ABB RobotStudio station: Train Assembling.rspag

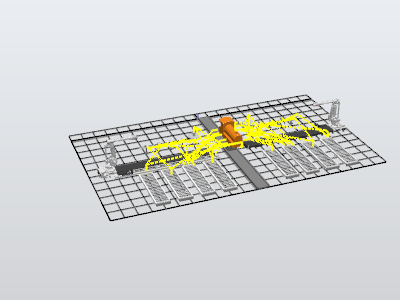
--- station ---
Station SimulationProject (saved by RobotStudio 24.3.10958.1)
Controller SimulationProject, task T_ROB2: task frame (RAPID world) sits at (6025, -9409.5, 384.5) mm, rotated rx 0 ry 0 rz 90 deg in the station
Controller SimulationProject, task T_ROB1: task frame (RAPID world) sits at (6025, -9409.5, 384.5) mm, rotated rx 0 ry 0 rz 90 deg in the station
Controller SimulationProject
  mechanical unit ROB_1: IRB6660_100_335__01_R, 6 joints, base frame (0, 0, 0) mm
  mechanical unit TRACK_1: IRBT6004_STD_0_0_8__04_R, 1 joints, base frame (0, 0, 0) mm
  mechanical unit ROB_2: IRB6660_100_335__01_L, 6 joints, base frame (19319, 50, 0) mm, rotated rx 0 ry 0 rz 180 deg
  mechanical unit TRACK_2: IRBT6004_STD_0_0_8__04_L, 1 joints, base frame (19319, 50, 0) mm, rotated rx 0 ry 0 rz 180 deg
Layout (positions relative to the parent item):
  - IRB6660_100_335__01_R [mechanism, from %ABB.RobotStudio.Models.IRB6660%\IRB6660_100_335_G_01.rslib] at (6025, -9409.5, 384.5) mm, rotated rx 0 ry 0 rz 90 deg; joint values [0, 0, 0, 0, 0.5236, 0] (rad or m)
  - IRBT6004_STD_0_0_8__04_R [mechanism] at (6500, -10000, 0) mm, rotated rx 0 ry 0 rz 90 deg; joint values [0] (rad or m)
      links: Base, Link1
  - IRB6660_100_335__01_L [mechanism, from %ABB.RobotStudio.Models.IRB6660%\IRB6660_100_335_G_01.rslib] at (5975, 9909.5, 384.5) mm, rotated rx 0 ry 0 rz -90 deg; joint values [0, 0, 0, 0, 0.5236, 0] (rad or m)
  - IRBT6004_STD_0_0_8__04_L [mechanism] at (5500, 10500, 0) mm, rotated rx 0 ry 0 rz -90 deg; joint values [0] (rad or m)
      links: Base, Link1
  - Train_Slider_Device [mechanism, from Tools\Train_Slider_Device.rslib] at (0, 0, 0) mm; joint values [5.8] (rad or m)
  - train_body [part] at (4625, 0, 1000) mm, rotated rx 90 ry 0 rz 90 deg, size 1000 x 1362.5 x 2750 mm
  - SC_Wheel_InFeeder_R [smart component]
      signals: DI FeedWheel
      connections:
        SC_Wheel_InFeeder_R.FeedWheel -> Source.Execute
        Source.Executed -> Queue.Enqueue
        PlaneSensor.SensorOut -> Queue.Dequeue
        Source.Copy => Queue.Back
        Queue.Front => PlaneSensor.SensedPart
    - LinearMover [smart component, from Components\LinearMover.rslib]
        properties: Object=Queue; Direction=[-1 0 0]; Speed=0.5; Reference=Global; ReferenceObject=(none)
    - Source [smart component, from Components\Source.rslib]
        properties: Source=Wheel_R; Copy=(none); Parent=(none); Position=[0 0 0]; Orientation=[0 0 0]; Transient=false; PhysicsBehavior=-1
    - Queue [smart component, from Components\Queue.rslib]
        properties: Back=(none); Front=(none); Queue={9305e1b5-9379-48da-9073-8e46354b7aa1};{06ef701b-e628-484b-9ba1-8a04eedeb4da};{5bc8af88-7b1d-4971-8da9-7f0ec308ea46};{a84a56de-22f5-4cb1-84ca-754a15d204a5};{2fea0387-14bd-40cc-a5c2-ab10d6d0a730};{1b48ac47-8c9f-46e7-a90e-52eff258e1c6};{a66a5858-2d20-4f19-907b-7c595a4e8944}; NumberOfObjects=1
    - PlaneSensor [smart component, from Components\PlaneSensor.rslib]
        properties: Origin=[7.64 -1.525 0.435]; Axis1=[0 0 0.2]; Axis2=[0 -0.9 0]; Tag=(none); SensedPart=(none)
      - _sensorPart_ [part], size 0 x 900 x 200 mm
    - InFeeder_R_1 [part] at (6500, -2000, 0) mm, size 4244 x 1170 x 435 mm
  - SC_Screws_InFeeder_R [smart component]
      signals: DI FeedScrews
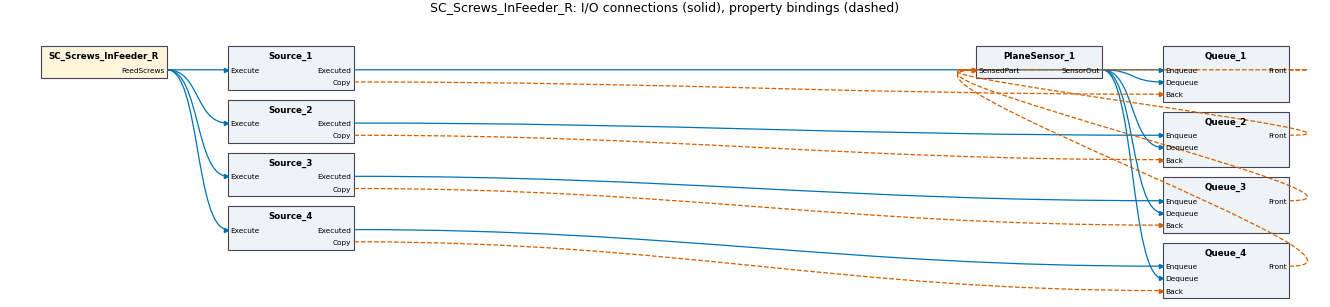
      connections:
        Source_1.Executed -> Queue_1.Enqueue
        Source_2.Executed -> Queue_2.Enqueue
        PlaneSensor_1.SensorOut -> Queue_1.Dequeue
        PlaneSensor_1.SensorOut -> Queue_2.Dequeue
        Source_3.Executed -> Queue_3.Enqueue
        Source_4.Executed -> Queue_4.Enqueue
        PlaneSensor_1.SensorOut -> Queue_3.Dequeue
        PlaneSensor_1.SensorOut -> Queue_4.Dequeue
        SC_Screws_InFeeder_R.FeedScrews -> Source_1.Execute
        SC_Screws_InFeeder_R.FeedScrews -> Source_2.Execute
        SC_Screws_InFeeder_R.FeedScrews -> Source_3.Execute
        SC_Screws_InFeeder_R.FeedScrews -> Source_4.Execute
        Source_1.Copy => Queue_1.Back
        Queue_1.Front => PlaneSensor_1.SensedPart
        Queue_2.Front => PlaneSensor_1.SensedPart
        Source_3.Copy => Queue_3.Back
        Source_4.Copy => Queue_4.Back
        Queue_3.Front => PlaneSensor_1.SensedPart
        Queue_4.Front => PlaneSensor_1.SensedPart
        Source_2.Copy => Queue_2.Back
    - InFeeder_R_2 [part] at (6500, -3700, 0) mm, size 4244 x 1170 x 435 mm
    - Source_1 [smart component, from Components\Source.rslib]
        properties: Source=Axel_pin_R_1; Copy=(none); Parent=(none); Position=[0 0 0]; Orientation=[0 0 0]; Transient=false; PhysicsBehavior=-1
    - Source_2 [smart component, from Components\Source.rslib]
        properties: Source=Axel_pin_R_2; Copy=(none); Parent=(none); Position=[0 0 0]; Orientation=[0 0 0]; Transient=false; PhysicsBehavior=-1
    - PlaneSensor_1 [smart component, from Components\PlaneSensor.rslib]
        properties: Origin=[7.64 -3.225 0.435]; Axis1=[0 -0.9 0]; Axis2=[0 0 0.2]; Tag=(none); SensedPart=(none)
      - _sensorPart_ [part], size 0 x 900 x 200 mm
    - Queue_1 [smart component, from Components\Queue.rslib]
        properties: Back=(none); Front=(none); Queue={97678c5a-5102-4407-a08a-453d650fad80};{250eec11-255d-4adc-99c6-b5c3b0be1ee0};{db8d0e62-9b7f-46e3-aee1-3fad0f8208f2};{3d23516b-ce9b-4da7-b7d3-33ea277e23c2};{336e8d4f-087f-4f39-84d7-9a0945deb51c};{844237c7-2bfb-4aaa-a27e-a2dee6dfaffc};{404c0b62-1524-42dd-8a4b-c3c094d3b07c}; NumberOfObjects=1
    - Queue_2 [smart component, from Components\Queue.rslib]
        properties: Back=(none); Front=(none); Queue={9e77e015-2590-4be3-ac1b-ed1168efcc9a};{9dcada67-6f7e-4e2e-9580-51d109b5ace8};{683b0bf4-25e8-4e74-bd3c-a3e39548362f}; NumberOfObjects=1
    - LinearMover_1 [smart component, from Components\LinearMover.rslib]
        properties: Object=Queue_1; Direction=[-1 0 0]; Speed=0.5; Reference=Global; ReferenceObject=(none)
    - LinearMover_2 [smart component, from Components\LinearMover.rslib]
        properties: Object=Queue_2; Direction=[-1 0 0]; Speed=0.5; Reference=Global; ReferenceObject=(none)
    - Source_3 [smart component, from Components\Source.rslib]
        properties: Source=Arm_pin_R_1; Copy=(none); Parent=(none); Position=[0 0 0]; Orientation=[0 0 0]; Transient=false; PhysicsBehavior=-1
    - Source_4 [smart component, from Components\Source.rslib]
        properties: Source=Arm_pin_R_2; Copy=(none); Parent=(none); Position=[0 0 0]; Orientation=[0 0 0]; Transient=false; PhysicsBehavior=-1
    - Queue_3 [smart component, from Components\Queue.rslib]
        properties: Back=(none); Front=(none); Queue={6ed0c4d3-6d0d-466e-bc0a-e55b9d8fea7f};{e0375d21-1e9d-4950-9f28-cd2b8b21485b};{fc4e43e4-3199-411d-82b8-a28eed2363bc};{00cf09c5-e1bb-4b7d-8b4f-d00f571ac579}; NumberOfObjects=1
    - Queue_4 [smart component, from Components\Queue.rslib]
        properties: Back=(none); Front=(none); Queue={3f8a16d5-ca92-48d5-91d9-dae51837d5b3};{1a52513d-85f7-411d-a240-a53d51e62410};{d2420088-7648-42ee-ace7-0250b97bbbd5};{92784dae-7df1-4f9f-a001-3219d183c38a}; NumberOfObjects=1
    - LinearMover_3 [smart component, from Components\LinearMover.rslib]
        properties: Object=Queue_3; Direction=[-1 0 0]; Speed=0.5; Reference=Global; ReferenceObject=(none)
    - LinearMover_4 [smart component, from Components\LinearMover.rslib]
        properties: Object=Queue_4; Direction=[-1 0 0]; Speed=0.5; Reference=Global; ReferenceObject=(none)
  - SC_Link_InFeeder_R [smart component]
      signals: DI FeedLink
      connections:
        PlaneSensor.SensorOut -> Queue.Dequeue
        Source.Executed -> Queue.Enqueue
        SC_Link_InFeeder_R.FeedLink -> Source.Execute
        Source.Copy => Queue.Back
        Queue.Front => PlaneSensor.SensedPart
    - InFeeder_R_3 [part] at (6500, -5400, 0) mm, size 4244 x 1170 x 435 mm
    - Source [smart component, from Components\Source.rslib]
        properties: Source=Link_R; Copy=(none); Parent=(none); Position=[0 0 0]; Orientation=[0 0 0]; Transient=false; PhysicsBehavior=-1
    - PlaneSensor [smart component, from Components\PlaneSensor.rslib]
        properties: Origin=[7.64 -4.925 0.435]; Axis1=[0 -0.9 0]; Axis2=[0 0 0.2]; Tag=(none); SensedPart=(none)
      - _sensorPart_ [part], size 0 x 900 x 200 mm
    - Queue [smart component, from Components\Queue.rslib]
        properties: Back=(none); Front=(none); Queue={c123ca29-f25a-4360-8441-2d47dce9963e};{cf207c4b-303d-438f-b968-cd8524d1301f};{72cfc707-1568-4af6-a666-0a4982008e72};{3a86617a-4034-4a56-87a3-25b6863a3576}; NumberOfObjects=1
    - LinearMover [smart component, from Components\LinearMover.rslib]
        properties: Object=Queue; Direction=[-1 0 0]; Speed=0.5; Reference=Global; ReferenceObject=(none)
  - SC_CowCatcher_InFeeder_R [smart component]
      signals: DI FeedCowCatcher
      connections:
        SC_CowCatcher_InFeeder_R.FeedCowCatcher -> Source_2.Execute
        Source_2.Executed -> Queue_2.Enqueue
        PlaneSensor_2.SensorOut -> Queue_2.Dequeue
        Source_2.Copy => Queue_2.Back
        Queue_2.Front => PlaneSensor_2.SensedPart
    - InFeeder_R_4 [part] at (6500, -7100, 0) mm, size 4244 x 1170 x 435 mm
    - LinearMover_2 [smart component, from Components\LinearMover.rslib]
        properties: Object=Queue_2; Direction=[-1 0 0]; Speed=0.5; Reference=Global; ReferenceObject=(none)
    - Queue_2 [smart component, from Components\Queue.rslib]
        properties: Back=(none); Front=(none); Queue={e25ade14-9086-4660-97fb-0c3a861d3266};{c5b81c7c-9b40-4532-81d4-bb342586ee21};{586fb502-498d-41ec-904b-685c852027eb}; NumberOfObjects=1
    - PlaneSensor_2 [smart component, from Components\PlaneSensor.rslib]
        properties: Origin=[7.64 -6.625 0.435]; Axis1=[0 -0.9 0]; Axis2=[0 0 0.2]; Tag=(none); SensedPart=(none)
      - _sensorPart_ [part], size 0 x 900 x 200 mm
    - Source_2 [smart component, from Components\Source.rslib]
        properties: Source=Cow_Catcher; Copy=(none); Parent=(none); Position=[0 0 0]; Orientation=[0 0 0]; Transient=false; PhysicsBehavior=-1
  - SC_Link_InFeeder_L [smart component] at (0, 11800, 0) mm
      signals: DI FeedLink_L
      connections:
        PlaneSensor.SensorOut -> Queue.Dequeue
        Source.Executed -> Queue.Enqueue
        SC_Link_InFeeder_L.FeedLink_L -> Source.Execute
        Source.Copy => Queue.Back
        Queue.Front => PlaneSensor.SensedPart
    - InFeeder_R_3 [part] at (6500, -5400, 0) mm, size 4244 x 1170 x 435 mm
    - Source [smart component, from Components\Source.rslib]
        properties: Source=Link_L; Copy=(none); Parent=(none); Position=[0 0 0]; Orientation=[0 0 0]; Transient=false; PhysicsBehavior=-1
    - PlaneSensor [smart component, from Components\PlaneSensor.rslib]
        properties: Origin=[7.64 -4.925 0.435]; Axis1=[0 -0.9 0]; Axis2=[0 0 0.2]; Tag=(none); SensedPart=(none)
      - _sensorPart_ [part], size 0 x 900 x 200 mm
    - Queue [smart component, from Components\Queue.rslib]
        properties: Back=(none); Front=(none); Queue={9254929b-264a-4685-b6a1-bce98a06c028};{c123ca29-f25a-4360-8441-2d47dce9963e};{cf207c4b-303d-438f-b968-cd8524d1301f};{4bafc17b-eeca-41b5-b438-7a43c40b0997};{fc8fee30-79e4-4b7d-9fd5-4bdb28a1c232};{eefd66af-0d0b-49de-8bd5-7017a8631d51};{a98b3633-ee36-4176-97fc-4a52fb264d0f}; NumberOfObjects=1
    - LinearMover [smart component, from Components\LinearMover.rslib]
        properties: Object=Queue; Direction=[-1 0 0]; Speed=0.5; Reference=Global; ReferenceObject=(none)
  - SC_Screws_InFeeder_L [smart component] at (0, 8400, 0) mm
      signals: DI FeedScrews_L
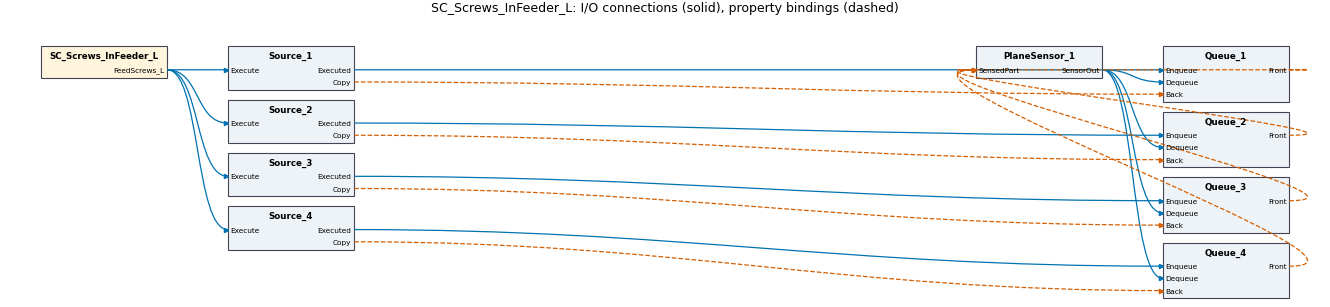
      connections:
        Source_1.Executed -> Queue_1.Enqueue
        Source_2.Executed -> Queue_2.Enqueue
        PlaneSensor_1.SensorOut -> Queue_1.Dequeue
        PlaneSensor_1.SensorOut -> Queue_2.Dequeue
        Source_3.Executed -> Queue_3.Enqueue
        Source_4.Executed -> Queue_4.Enqueue
        PlaneSensor_1.SensorOut -> Queue_3.Dequeue
        PlaneSensor_1.SensorOut -> Queue_4.Dequeue
        SC_Screws_InFeeder_L.FeedScrews_L -> Source_1.Execute
        SC_Screws_InFeeder_L.FeedScrews_L -> Source_2.Execute
        SC_Screws_InFeeder_L.FeedScrews_L -> Source_3.Execute
        SC_Screws_InFeeder_L.FeedScrews_L -> Source_4.Execute
        Source_1.Copy => Queue_1.Back
        Queue_1.Front => PlaneSensor_1.SensedPart
        Queue_2.Front => PlaneSensor_1.SensedPart
        Source_3.Copy => Queue_3.Back
        Source_4.Copy => Queue_4.Back
        Queue_3.Front => PlaneSensor_1.SensedPart
        Queue_4.Front => PlaneSensor_1.SensedPart
        Source_2.Copy => Queue_2.Back
    - InFeeder_R_2 [part] at (6500, -3700, 0) mm, size 4244 x 1170 x 435 mm
    - Source_1 [smart component, from Components\Source.rslib]
        properties: Source=Axel_pin_L_1; Copy=(none); Parent=(none); Position=[0 0 0]; Orientation=[0 0 0]; Transient=false; PhysicsBehavior=-1
    - Source_2 [smart component, from Components\Source.rslib]
        properties: Source=Axel_pin_L_2; Copy=(none); Parent=(none); Position=[0 0 0]; Orientation=[0 0 0]; Transient=false; PhysicsBehavior=-1
    - PlaneSensor_1 [smart component, from Components\PlaneSensor.rslib]
        properties: Origin=[7.64 -3.225 0.435]; Axis1=[0 -0.9 0]; Axis2=[0 0 0.2]; Tag=(none); SensedPart=(none)
      - _sensorPart_ [part], size 0 x 900 x 200 mm
    - Queue_1 [smart component, from Components\Queue.rslib]
        properties: Back=(none); Front=(none); Queue={14a08090-38d6-472e-a98c-ca0218ab0c7a};{97678c5a-5102-4407-a08a-453d650fad80};{250eec11-255d-4adc-99c6-b5c3b0be1ee0};{db8d0e62-9b7f-46e3-aee1-3fad0f8208f2};{2b439d8e-8bb8-4235-883a-6f3a83c8853b};{c95d82af-f454-4449-b05f-7ed691318b29};{bee60a8c-c6b8-489c-bade-25b0cdd1ce0b};{754e9011-9557-4989-aa10-6dc2dc1ac779}; NumberOfObjects=1
    - Queue_2 [smart component, from Components\Queue.rslib]
        properties: Back=(none); Front=(none); Queue=; NumberOfObjects=0
    - LinearMover_1 [smart component, from Components\LinearMover.rslib]
        properties: Object=Queue_1; Direction=[-1 0 0]; Speed=0.5; Reference=Global; ReferenceObject=(none)
    - LinearMover_2 [smart component, from Components\LinearMover.rslib]
        properties: Object=Queue_2; Direction=[-1 0 0]; Speed=0.5; Reference=Global; ReferenceObject=(none)
    - Source_3 [smart component, from Components\Source.rslib]
        properties: Source=Arm_pin_L_1; Copy=(none); Parent=(none); Position=[0 0 0]; Orientation=[0 0 0]; Transient=false; PhysicsBehavior=-1
    - Source_4 [smart component, from Components\Source.rslib]
        properties: Source=Arm_pin_L_2; Copy=(none); Parent=(none); Position=[0 0 0]; Orientation=[0 0 0]; Transient=false; PhysicsBehavior=-1
    - Queue_3 [smart component, from Components\Queue.rslib]
        properties: Back=(none); Front=(none); Queue={ed4f623c-c085-4233-b9e7-8bb17121263c};{7df952f9-3ef9-4a6d-b65d-53123e49cebe};{7d5f55dc-9dc7-46c2-bf9a-09a703fb0915};{9adc3934-4715-46cc-a34c-30ea8ea2b250};{ca0e7fb5-f50a-45a6-838f-04012fdc7c55}; NumberOfObjects=1
    - Queue_4 [smart component, from Components\Queue.rslib]
        properties: Back=(none); Front=(none); Queue={0f597643-c704-410c-a7ca-8884bd8ca932};{edcab222-0b96-4825-ae17-e599e194de34};{f3ecc827-54de-4d18-b44b-cadbdeb3097c};{053afdf7-4801-444a-88ee-4a240900a0be};{0f677b95-c554-4bb8-81c5-1595ff83ef41}; NumberOfObjects=1
    - LinearMover_3 [smart component, from Components\LinearMover.rslib]
        properties: Object=Queue_3; Direction=[-1 0 0]; Speed=0.5; Reference=Global; ReferenceObject=(none)
    - LinearMover_4 [smart component, from Components\LinearMover.rslib]
        properties: Object=Queue_4; Direction=[-1 0 0]; Speed=0.5; Reference=Global; ReferenceObject=(none)
  - SC_Stack_InFeeder_L [smart component] at (0, 15200, 0) mm
      signals: DI FeedStack
      connections:
        Source_2.Executed -> Queue_2.Enqueue
        PlaneSensor_2.SensorOut -> Queue_2.Dequeue
        SC_Stack_InFeeder_L.FeedStack -> Source_2.Execute
        Source_2.Copy => Queue_2.Back
        Queue_2.Front => PlaneSensor_2.SensedPart
    - InFeeder_R_4 [part] at (6500, -7100, 0) mm, size 4244 x 1170 x 435 mm
    - LinearMover_2 [smart component, from Components\LinearMover.rslib]
        properties: Object=Queue_2; Direction=[-1 0 0]; Speed=0.5; Reference=Global; ReferenceObject=(none)
    - Queue_2 [smart component, from Components\Queue.rslib]
        properties: Back=(none); Front=(none); Queue={08baaac3-cf0c-443c-8ac5-ab6bfb04582b};{e25ade14-9086-4660-97fb-0c3a861d3266};{a7b411b6-9305-4ad5-91da-d1a51fd8feb1};{f2907e09-aa18-4079-bd41-b284c3e6ed90};{4df58e7f-3ce5-4aae-ac92-7c7a7f14669e};{580da0eb-0ea4-4e5a-8dee-4f1589a54273}; NumberOfObjects=1
    - PlaneSensor_2 [smart component, from Components\PlaneSensor.rslib]
        properties: Origin=[7.64 -6.625 0.435]; Axis1=[0 -0.9 0]; Axis2=[0 0 0.2]; Tag=(none); SensedPart=(none)
      - _sensorPart_ [part], size 0 x 900 x 200 mm
    - Source_2 [smart component, from Components\Source.rslib]
        properties: Source=Stack_tutorial; Copy=(none); Parent=(none); Position=[0 0 0]; Orientation=[0 0 0]; Transient=false; PhysicsBehavior=-1
  - SC_Wheel_InFeeder_L [smart component] at (0, 5000, 0) mm
      signals: DI FeedWheel_L
      connections:
        Source.Executed -> Queue.Enqueue
        PlaneSensor.SensorOut -> Queue.Dequeue
        SC_Wheel_InFeeder_L.FeedWheel_L -> Source.Execute
        Source.Copy => Queue.Back
        Queue.Front => PlaneSensor.SensedPart
    - LinearMover [smart component, from Components\LinearMover.rslib]
        properties: Object=Queue; Direction=[-1 0 0]; Speed=0.5; Reference=Global; ReferenceObject=(none)
    - Source [smart component, from Components\Source.rslib]
        properties: Source=Wheel_L; Copy=(none); Parent=(none); Position=[0 0 0]; Orientation=[0 0 0]; Transient=false; PhysicsBehavior=-1
    - Queue [smart component, from Components\Queue.rslib]
        properties: Back=(none); Front=(none); Queue={f792bd7d-59b8-452e-8621-f4f9bd52dab3};{60f8df29-37bb-424b-bc17-7874fedc1897};{9305e1b5-9379-48da-9073-8e46354b7aa1};{06ef701b-e628-484b-9ba1-8a04eedeb4da};{5bc8af88-7b1d-4971-8da9-7f0ec308ea46};{2c83ba85-32fa-4865-9bd8-e969231fd573};{529ee98c-f03b-47d6-93bf-629f2e0b32d3};{d39da287-2192-4b0a-90db-445a384171d5};{c893a77d-bff1-42fa-8d0e-c2cc12e39c3c}; NumberOfObjects=1
    - PlaneSensor [smart component, from Components\PlaneSensor.rslib]
        properties: Origin=[7.64 -1.525 0.435]; Axis1=[0 0 0.2]; Axis2=[0 -0.9 0]; Tag=(none); SensedPart=(none)
      - _sensorPart_ [part], size 0 x 900 x 200 mm
    - InFeeder_R_1 [part] at (6500, -2000, 0) mm, size 4244 x 1170 x 435 mm
  - Tool_Holder_B_R_1 [part, from Tools\Tool_Holder_B.rslib] at (4000, -2000, 0) mm
  - Tool_Holder_S_R_2 [part, from Tools\Tool_Holder_S.rslib] at (4000, -3000, 0) mm
  - Tool_Holder_S_R_3 [part, from Tools\Tool_Holder_S.rslib] at (4000, -4000, 0) mm
  - Tool_Holder_S_R_4 [part, from Tools\Tool_Holder_S.rslib] at (4000, -5000, 0) mm
  - Tool_Holder_M_R_5 [part, from Tools\Tool_Holder_M.rslib] at (4000, -6000, 0) mm
  - ArmPinTool_R [mechanism, from Tools\ArmPinTool.rslib] at (4200, -3900, 800) mm, rotated rx 180 ry 0 rz 0 deg
  - AxelPinTool_R [mechanism, from Tools\AxelPinTool.rslib] at (4200, -2900, 800) mm, rotated rx 180 ry 0 rz 0 deg
  - CowCatcherTool_R [mechanism, from Tools\CowCatcherTool.rslib] at (4220, -4900, 800) mm, rotated rx 180 ry 0 rz 180 deg
  - WheelTool_R [mechanism, from Tools\WheelTool.rslib] at (4050, -1900, 1130) mm, rotated rx 180 ry 0 rz 180 deg
  - Wheel_R [part], size 1122.9 x 1119.7 x 250 mm
  - Link_R [part], size 1937.5 x 186.8 x 62.5 mm
  - Cow_Catcher [part], size 562.5 x 900 x 375 mm
  - Arm_pin_R_2 [part], size 162.5 x 126 x 125.8 mm
  - Arm_pin_R_1 [part], size 162.5 x 126 x 125.8 mm
  - Tool_Holder_B_L_1 [part, from Tools\Tool_Holder_B.rslib] at (3500, 3000, 0) mm
  - Tool_Holder_S_L_2 [part, from Tools\Tool_Holder_S.rslib] at (3500, 4000, 0) mm
  - Tool_Holder_S_L_3 [part, from Tools\Tool_Holder_S.rslib] at (3500, 5000, 0) mm
  - Tool_Holder_S_L_4 [part, from Tools\Tool_Holder_S.rslib] at (3500, 6000, 0) mm
  - Tool_Holder_M_L_5 [part, from Tools\Tool_Holder_M.rslib] at (3500, 7000, 0) mm
  - WheelTool_L [mechanism, from Tools\WheelTool.rslib] at (3550, 3100, 1130) mm, rotated rx 180 ry 0 rz 180 deg
  - StackTool [mechanism, from Tools\StackTool.rslib] at (3700, 6100, 800) mm, rotated rx 180 ry 0 rz 0 deg
  - AxelPinTool_L [mechanism, from Tools\AxelPinTool.rslib] at (3700, 4100, 800) mm, rotated rx 180 ry 0 rz 0 deg
  - ArmPinTool_L [mechanism, from Tools\ArmPinTool.rslib] at (3700, 5100, 800) mm, rotated rx 180 ry 0 rz 0 deg
  - Wheel_L [part], size 1122.9 x 1119.7 x 250 mm
  - Link_L [part], size 1937.5 x 186.8 x 62.5 mm
  - Axel_pin_L_1 [part], size 562.7 x 211 x 211 mm
  - Axel_pin_L_2 [part], size 562.7 x 211 x 211 mm
  - Arm_pin_L_1 [part], size 162.5 x 126 x 125.8 mm
  - Arm_pin_L_2 [part], size 162.5 x 126 x 125.8 mm
  - Stack_tutorial [part], size 625 x 623.8 x 875 mm
  - Axel_pin_R_2 [part], size 562.7 x 211 x 211 mm
  - Axel_pin_R_1 [part], size 562.7 x 211 x 211 mm
  - LinkTool_R [mechanism, from Tools\LinkTool.rslib] at (4199.56, -5900, 800) mm, rotated rx -180 ry 0 rz 0 deg
  - LinkTool_L [mechanism, from Tools\LinkTool.rslib] at (3700, 7100, 800) mm, rotated rx 180 ry 0 rz 0 deg
Attachment: IRB6660_100_335__01_R is attached to IRBT6004_STD_0_0_8__04_R / Link1
Attachment: IRB6660_100_335__01_L is attached to IRBT6004_STD_0_0_8__04_L / Link1
Attachment: Train_Slider_Device is attached to train_body
EventTableEntry 6243: ActivationMode=2, Cyclic=false, Group=, Trigger=doWheelTool 6244, Actions=[EventTableActionAttach 6245], Comment=
EventTableTriggerIO 6244: Operator=0, IOValue=[1], IRC5Controller=? -1, SignalSource=SimulationProject 3637
EventTableActionAttach 6245: MountObject=false, FlangeIndext=0, FindNearest=false, AttachmentParent=IRB6660_100_335__01_R 3560, AttachmentChild=WheelTool_R 5965, Offset=[X=1, Y=0, Z=0, W=0, X=0, Y=1, Z=0, W=0, X=0, Y=0, Z=1, W=0, X=0, Y=0, Z=0, W=1]
EventTableEntry 6246: ActivationMode=2, Cyclic=false, Group=, Trigger=doWheelTool 6247, Actions=[EventTableActionDetach 6248], Comment=
EventTableTriggerIO 6247: Operator=0, IOValue=[0], IRC5Controller=? -1, SignalSource=SimulationProject 3637
EventTableActionDetach 6248: AttachmentParent=IRB6660_100_335__01_R 3560, AttachmentChild=WheelTool_R 5965
EventTableEntry 6249: ActivationMode=2, Cyclic=false, Group=, Trigger=doWheel 6250, Actions=[EventTableActionAttach 6251], Comment=
EventTableTriggerIO 6250: Operator=0, IOValue=[1], IRC5Controller=? -1, SignalSource=SimulationProject 3637
EventTableActionAttach 6251: MountObject=false, FlangeIndext=0, FindNearest=true, AttachmentParent=WheelTool_R 5965, AttachmentChild=? -1, Offset=[X=1, Y=0, Z=0, W=0, X=0, Y=1, Z=0, W=0, X=0, Y=0, Z=1, W=0, X=0, Y=0, Z=0, W=1]
EventTableTriggerIO 6346: Operator=0, IOValue=[1], IRC5Controller=? -1, SignalSource=SimulationProject 3637
EventTableTriggerIO 6347: Operator=0, IOValue=[1], IRC5Controller=? -1, SignalSource=SimulationProject 3637
EventTableTriggerIO 6348: Operator=0, IOValue=[1], IRC5Controller=? -1, SignalSource=SimulationProject 3637
EventTableTriggerIO 6349: Operator=0, IOValue=[1], IRC5Controller=? -1, SignalSource=SimulationProject 3637
EventTableTriggerIO 6350: Operator=0, IOValue=[0], IRC5Controller=? -1, SignalSource=SimulationProject 3637
EventTableTriggerIO 6351: Operator=0, IOValue=[0], IRC5Controller=? -1, SignalSource=SimulationProject 3637
EventTableTriggerIO 6352: Operator=0, IOValue=[0], IRC5Controller=? -1, SignalSource=SimulationProject 3637
EventTableTriggerIO 6353: Operator=0, IOValue=[0], IRC5Controller=? -1, SignalSource=SimulationProject 3637
EventTableTriggerIO 6354: Operator=0, IOValue=[1], IRC5Controller=? -1, SignalSource=SimulationProject 3637
EventTableTriggerIO 6355: Operator=0, IOValue=[1], IRC5Controller=? -1, SignalSource=SimulationProject 3637
EventTableTriggerIO 6356: Operator=0, IOValue=[1], IRC5Controller=? -1, SignalSource=SimulationProject 3637
EventTableTriggerIO 6357: Operator=0, IOValue=[1], IRC5Controller=? -1, SignalSource=SimulationProject 3637
EventTableEntry 6358: ActivationMode=2, Cyclic=false, Group=, Trigger=doWheel 6359, Actions=[EventTableActionDetach 6360], Comment=
EventTableTriggerIO 6359: Operator=0, IOValue=[0], IRC5Controller=? -1, SignalSource=SimulationProject 3637
EventTableActionDetach 6360: AttachmentParent=WheelTool_R 5965, AttachmentChild=? -1
EventTableTriggerIO 6361: Operator=0, IOValue=[0], IRC5Controller=? -1, SignalSource=SimulationProject 3637
EventTableTriggerIO 6362: Operator=0, IOValue=[0], IRC5Controller=? -1, SignalSource=SimulationProject 3637
EventTableTriggerIO 6363: Operator=0, IOValue=[0], IRC5Controller=? -1, SignalSource=SimulationProject 3637
EventTableTriggerIO 6364: Operator=0, IOValue=[0], IRC5Controller=? -1, SignalSource=SimulationProject 3637
EventTableTriggerIO 6724: Operator=0, IOValue=[1], IRC5Controller=? -1, SignalSource=SimulationProject 3637
EventTableTriggerIO 6725: Operator=0, IOValue=[0], IRC5Controller=? -1, SignalSource=SimulationProject 3637
EventTableTriggerIO 6726: Operator=0, IOValue=[1], IRC5Controller=? -1, SignalSource=SimulationProject 3637
EventTableTriggerIO 6727: Operator=0, IOValue=[0], IRC5Controller=? -1, SignalSource=SimulationProject 3637
EventTableTriggerIO 6969: Operator=0, IOValue=[1], IRC5Controller=? -1, SignalSource=SimulationProject 3637
EventTableTriggerIO 6970: Operator=0, IOValue=[0], IRC5Controller=? -1, SignalSource=SimulationProject 3637
EventTableTriggerIO 6971: Operator=0, IOValue=[1], IRC5Controller=? -1, SignalSource=SimulationProject 3637
EventTableTriggerIO 6972: Operator=0, IOValue=[0], IRC5Controller=? -1, SignalSource=SimulationProject 3637
EventTableEntry 6973: ActivationMode=2, Cyclic=false, Group=, Trigger=doAxelTool 6974, Actions=[EventTableActionAttach 6975], Comment=
EventTableTriggerIO 6974: Operator=0, IOValue=[1], IRC5Controller=? -1, SignalSource=SimulationProject 3637
EventTableActionAttach 6975: MountObject=false, FlangeIndext=0, FindNearest=false, AttachmentParent=IRB6660_100_335__01_R 3560, AttachmentChild=AxelPinTool_R 5956, Offset=[X=1, Y=0, Z=0, W=0, X=0, Y=1, Z=0, W=0, X=0, Y=0, Z=1, W=0, X=0, Y=0, Z=0, W=1]
EventTableEntry 6976: ActivationMode=2, Cyclic=false, Group=, Trigger=doAxelTool 6977, Actions=[EventTableActionDetach 6978], Comment=
EventTableTriggerIO 6977: Operator=0, IOValue=[0], IRC5Controller=? -1, SignalSource=SimulationProject 3637
EventTableActionDetach 6978: AttachmentParent=IRB6660_100_335__01_R 3560, AttachmentChild=AxelPinTool_R 5956
EventTableEntry 6979: ActivationMode=2, Cyclic=false, Group=, Trigger=doAxel 6980, Actions=[EventTableActionAttach 6981], Comment=
EventTableTriggerIO 6980: Operator=0, IOValue=[1], IRC5Controller=? -1, SignalSource=SimulationProject 3637
EventTableActionAttach 6981: MountObject=false, FlangeIndext=0, FindNearest=true, AttachmentParent=AxelPinTool_R 5956, AttachmentChild=? -1, Offset=[X=1, Y=0, Z=0, W=0, X=0, Y=1, Z=0, W=0, X=0, Y=0, Z=1, W=0, X=0, Y=0, Z=0, W=1]
EventTableEntry 6982: ActivationMode=2, Cyclic=false, Group=, Trigger=doAxel 6983, Actions=[EventTableActionDetach 6984], Comment=
EventTableTriggerIO 6983: Operator=0, IOValue=[0], IRC5Controller=? -1, SignalSource=SimulationProject 3637
EventTableActionDetach 6984: AttachmentParent=AxelPinTool_R 5956, AttachmentChild=? -1
EventTableTriggerIO 7195: Operator=0, IOValue=[1], IRC5Controller=? -1, SignalSource=SimulationProject 3637
EventTableTriggerIO 7196: Operator=0, IOValue=[1], IRC5Controller=? -1, SignalSource=SimulationProject 3637
EventTableTriggerIO 7197: Operator=0, IOValue=[0], IRC5Controller=? -1, SignalSource=SimulationProject 3637
EventTableTriggerIO 7198: Operator=0, IOValue=[0], IRC5Controller=? -1, SignalSource=SimulationProject 3637
EventTableTriggerIO 7199: Operator=0, IOValue=[1], IRC5Controller=? -1, SignalSource=SimulationProject 3637
EventTableTriggerIO 7200: Operator=0, IOValue=[1], IRC5Controller=? -1, SignalSource=SimulationProject 3637
EventTableTriggerIO 7201: Operator=0, IOValue=[0], IRC5Controller=? -1, SignalSource=SimulationProject 3637
EventTableTriggerIO 7202: Operator=0, IOValue=[0], IRC5Controller=? -1, SignalSource=SimulationProject 3637
EventTableTriggerIO 7203: Operator=0, IOValue=[1], IRC5Controller=? -1, SignalSource=SimulationProject 3637
EventTableTriggerIO 7204: Operator=0, IOValue=[1], IRC5Controller=? -1, SignalSource=SimulationProject 3637
EventTableTriggerIO 7205: Operator=0, IOValue=[0], IRC5Controller=? -1, SignalSource=SimulationProject 3637
EventTableTriggerIO 7206: Operator=0, IOValue=[0], IRC5Controller=? -1, SignalSource=SimulationProject 3637
EventTableTriggerIO 7207: Operator=0, IOValue=[1], IRC5Controller=? -1, SignalSource=SimulationProject 3637
EventTableTriggerIO 7208: Operator=0, IOValue=[1], IRC5Controller=? -1, SignalSource=SimulationProject 3637
EventTableTriggerIO 7209: Operator=0, IOValue=[0], IRC5Controller=? -1, SignalSource=SimulationProject 3637
EventTableTriggerIO 7210: Operator=0, IOValue=[0], IRC5Controller=? -1, SignalSource=SimulationProject 3637
EventTableEntry 7533: ActivationMode=2, Cyclic=false, Group=, Trigger=doLinkTool 7534, Actions=[EventTableActionAttach 7535], Comment=
EventTableTriggerIO 7534: Operator=0, IOValue=[1], IRC5Controller=? -1, SignalSource=SimulationProject 3637
EventTableActionAttach 7535: MountObject=false, FlangeIndext=0, FindNearest=false, AttachmentParent=IRB6660_100_335__01_R 3560, AttachmentChild=LinkTool_R 7465, Offset=[X=1, Y=0, Z=0, W=0, X=0, Y=1, Z=0, W=0, X=0, Y=0, Z=1, W=0, X=0, Y=0, Z=0, W=1]
EventTableEntry 7536: ActivationMode=2, Cyclic=false, Group=, Trigger=doLinkTool 7537, Actions=[EventTableActionDetach 7538], Comment=
EventTableTriggerIO 7537: Operator=0, IOValue=[0], IRC5Controller=? -1, SignalSource=SimulationProject 3637
EventTableActionDetach 7538: AttachmentParent=IRB6660_100_335__01_R 3560, AttachmentChild=LinkTool_R 7465
EventTableEntry 7539: ActivationMode=2, Cyclic=false, Group=, Trigger=doLink 7540, Actions=[EventTableActionAttach 7541], Comment=
EventTableTriggerIO 7540: Operator=0, IOValue=[1], IRC5Controller=? -1, SignalSource=SimulationProject 3637
EventTableActionAttach 7541: MountObject=false, FlangeIndext=0, FindNearest=true, AttachmentParent=LinkTool_R 7465, AttachmentChild=? -1, Offset=[X=1, Y=0, Z=0, W=0, X=0, Y=1, Z=0, W=0, X=0, Y=0, Z=1, W=0, X=0, Y=0, Z=0, W=1]
EventTableEntry 7542: ActivationMode=2, Cyclic=false, Group=, Trigger=doLink 7543, Actions=[EventTableActionDetach 7544], Comment=
EventTableTriggerIO 7543: Operator=0, IOValue=[0], IRC5Controller=? -1, SignalSource=SimulationProject 3637
EventTableActionDetach 7544: AttachmentParent=LinkTool_R 7465, AttachmentChild=? -1
EventTableTriggerIO 7701: Operator=0, IOValue=[1], IRC5Controller=? -1, SignalSource=SimulationProject 3637
EventTableTriggerIO 7702: Operator=0, IOValue=[0], IRC5Controller=? -1, SignalSource=SimulationProject 3637
EventTableTriggerIO 7703: Operator=0, IOValue=[1], IRC5Controller=? -1, SignalSource=SimulationProject 3637
EventTableTriggerIO 7704: Operator=0, IOValue=[0], IRC5Controller=? -1, SignalSource=SimulationProject 3637
EventTableTriggerIO 7705: Operator=0, IOValue=[1], IRC5Controller=? -1, SignalSource=SimulationProject 3637
EventTableTriggerIO 7706: Operator=0, IOValue=[0], IRC5Controller=? -1, SignalSource=SimulationProject 3637
EventTableTriggerIO 7707: Operator=0, IOValue=[1], IRC5Controller=? -1, SignalSource=SimulationProject 3637
EventTableTriggerIO 7708: Operator=0, IOValue=[0], IRC5Controller=? -1, SignalSource=SimulationProject 3637
EventTableTriggerIO 7709: Operator=0, IOValue=[1], IRC5Controller=? -1, SignalSource=SimulationProject 3637
EventTableTriggerIO 7710: Operator=0, IOValue=[0], IRC5Controller=? -1, SignalSource=SimulationProject 3637
EventTableTriggerIO 7711: Operator=0, IOValue=[1], IRC5Controller=? -1, SignalSource=SimulationProject 3637
EventTableTriggerIO 7712: Operator=0, IOValue=[0], IRC5Controller=? -1, SignalSource=SimulationProject 3637
EventTableEntry 8043: ActivationMode=2, Cyclic=false, Group=, Trigger=doArmTool 8044, Actions=[EventTableActionAttach 8045], Comment=
EventTableTriggerIO 8044: Operator=0, IOValue=[1], IRC5Controller=? -1, SignalSource=SimulationProject 3637
EventTableActionAttach 8045: MountObject=false, FlangeIndext=0, FindNearest=false, AttachmentParent=IRB6660_100_335__01_R 3560, AttachmentChild=ArmPinTool_R 5953, Offset=[X=1, Y=0, Z=0, W=0, X=0, Y=1, Z=0, W=0, X=0, Y=0, Z=1, W=0, X=0, Y=0, Z=0, W=1]
EventTableEntry 8046: ActivationMode=2, Cyclic=false, Group=, Trigger=doArmTool 8047, Actions=[EventTableActionDetach 8048], Comment=
EventTableTriggerIO 8047: Operator=0, IOValue=[0], IRC5Controller=? -1, SignalSource=SimulationProject 3637
EventTableActionDetach 8048: AttachmentParent=IRB6660_100_335__01_R 3560, AttachmentChild=ArmPinTool_R 5953
EventTableEntry 8049: ActivationMode=2, Cyclic=false, Group=, Trigger=doArm 8050, Actions=[EventTableActionAttach 8051], Comment=
EventTableTriggerIO 8050: Operator=0, IOValue=[1], IRC5Controller=? -1, SignalSource=SimulationProject 3637
EventTableActionAttach 8051: MountObject=false, FlangeIndext=0, FindNearest=true, AttachmentParent=ArmPinTool_R 5953, AttachmentChild=? -1, Offset=[X=1, Y=0, Z=0, W=0, X=0, Y=1, Z=0, W=0, X=0, Y=0, Z=1, W=0, X=0, Y=0, Z=0, W=1]
EventTableEntry 8052: ActivationMode=2, Cyclic=false, Group=, Trigger=doArm 8053, Actions=[EventTableActionDetach 8054], Comment=
EventTableTriggerIO 8053: Operator=0, IOValue=[0], IRC5Controller=? -1, SignalSource=SimulationProject 3637
EventTableActionDetach 8054: AttachmentParent=ArmPinTool_R 5953, AttachmentChild=? -1
EventTableTriggerIO 8264: Operator=0, IOValue=[1], IRC5Controller=? -1, SignalSource=SimulationProject 3637
EventTableTriggerIO 8265: Operator=0, IOValue=[0], IRC5Controller=? -1, SignalSource=SimulationProject 3637
EventTableTriggerIO 8266: Operator=0, IOValue=[1], IRC5Controller=? -1, SignalSource=SimulationProject 3637
EventTableTriggerIO 8267: Operator=0, IOValue=[0], IRC5Controller=? -1, SignalSource=SimulationProject 3637
EventTableTriggerIO 8268: Operator=0, IOValue=[1], IRC5Controller=? -1, SignalSource=SimulationProject 3637
EventTableTriggerIO 8269: Operator=0, IOValue=[0], IRC5Controller=? -1, SignalSource=SimulationProject 3637
EventTableTriggerIO 8270: Operator=0, IOValue=[1], IRC5Controller=? -1, SignalSource=SimulationProject 3637
EventTableTriggerIO 8271: Operator=0, IOValue=[0], IRC5Controller=? -1, SignalSource=SimulationProject 3637
EventTableTriggerIO 8272: Operator=0, IOValue=[1], IRC5Controller=? -1, SignalSource=SimulationProject 3637
EventTableTriggerIO 8273: Operator=0, IOValue=[0], IRC5Controller=? -1, SignalSource=SimulationProject 3637
EventTableTriggerIO 8274: Operator=0, IOValue=[1], IRC5Controller=? -1, SignalSource=SimulationProject 3637
EventTableTriggerIO 8275: Operator=0, IOValue=[0], IRC5Controller=? -1, SignalSource=SimulationProject 3637
EventTableTriggerIO 8276: Operator=0, IOValue=[1], IRC5Controller=? -1, SignalSource=SimulationProject 3637
EventTableTriggerIO 8277: Operator=0, IOValue=[0], IRC5Controller=? -1, SignalSource=SimulationProject 3637
EventTableTriggerIO 8278: Operator=0, IOValue=[1], IRC5Controller=? -1, SignalSource=SimulationProject 3637
EventTableTriggerIO 8279: Operator=0, IOValue=[0], IRC5Controller=? -1, SignalSource=SimulationProject 3637
EventTableTriggerIO 8576: Operator=0, IOValue=[1], IRC5Controller=? -1, SignalSource=SimulationProject 3637
EventTableTriggerIO 8577: Operator=0, IOValue=[0], IRC5Controller=? -1, SignalSource=SimulationProject 3637
EventTableTriggerIO 8578: Operator=0, IOValue=[1], IRC5Controller=? -1, SignalSource=SimulationProject 3637
EventTableTriggerIO 8579: Operator=0, IOValue=[0], IRC5Controller=? -1, SignalSource=SimulationProject 3637
EventTableTriggerIO 8580: Operator=0, IOValue=[1], IRC5Controller=? -1, SignalSource=SimulationProject 3637
EventTableTriggerIO 8581: Operator=0, IOValue=[0], IRC5Controller=? -1, SignalSource=SimulationProject 3637
EventTableTriggerIO 8582: Operator=0, IOValue=[1], IRC5Controller=? -1, SignalSource=SimulationProject 3637
EventTableTriggerIO 8583: Operator=0, IOValue=[0], IRC5Controller=? -1, SignalSource=SimulationProject 3637
EventTableTriggerIO 8584: Operator=0, IOValue=[1], IRC5Controller=? -1, SignalSource=SimulationProject 3637
EventTableTriggerIO 8585: Operator=0, IOValue=[0], IRC5Controller=? -1, SignalSource=SimulationProject 3637
EventTableTriggerIO 8586: Operator=0, IOValue=[1], IRC5Controller=? -1, SignalSource=SimulationProject 3637
EventTableTriggerIO 8587: Operator=0, IOValue=[0], IRC5Controller=? -1, SignalSource=SimulationProject 3637
EventTableTriggerIO 8588: Operator=0, IOValue=[1], IRC5Controller=? -1, SignalSource=SimulationProject 3637
EventTableTriggerIO 8589: Operator=0, IOValue=[0], IRC5Controller=? -1, SignalSource=SimulationProject 3637
EventTableTriggerIO 8590: Operator=0, IOValue=[1], IRC5Controller=? -1, SignalSource=SimulationProject 3637
EventTableTriggerIO 8591: Operator=0, IOValue=[0], IRC5Controller=? -1, SignalSource=SimulationProject 3637
EventTableEntry 8592: ActivationMode=2, Cyclic=false, Group=, Trigger=doCowTool 8593, Actions=[EventTableActionAttach 8594], Comment=
EventTableTriggerIO 8593: Operator=0, IOValue=[1], IRC5Controller=? -1, SignalSource=SimulationProject 3637
EventTableActionAttach 8594: MountObject=false, FlangeIndext=0, FindNearest=false, AttachmentParent=IRB6660_100_335__01_R 3560, AttachmentChild=CowCatcherTool_R 5959, Offset=[X=1, Y=0, Z=0, W=0, X=0, Y=1, Z=0, W=0, X=0, Y=0, Z=1, W=0, X=0, Y=0, Z=0, W=1]
EventTableEntry 8595: ActivationMode=2, Cyclic=false, Group=, Trigger=doCowTool 8596, Actions=[EventTableActionDetach 8597], Comment=
EventTableTriggerIO 8596: Operator=0, IOValue=[0], IRC5Controller=? -1, SignalSource=SimulationProject 3637
EventTableActionDetach 8597: AttachmentParent=IRB6660_100_335__01_R 3560, AttachmentChild=CowCatcherTool_R 5959
EventTableEntry 8598: ActivationMode=2, Cyclic=false, Group=, Trigger=doCow 8599, Actions=[EventTableActionAttach 8600], Comment=
EventTableTriggerIO 8599: Operator=0, IOValue=[1], IRC5Controller=? -1, SignalSource=SimulationProject 3637
EventTableActionAttach 8600: MountObject=false, FlangeIndext=0, FindNearest=true, AttachmentParent=CowCatcherTool_R 5959, AttachmentChild=? -1, Offset=[X=1, Y=0, Z=0, W=0, X=0, Y=1, Z=0, W=0, X=0, Y=0, Z=1, W=0, X=0, Y=0, Z=0, W=1]
EventTableEntry 8601: ActivationMode=2, Cyclic=false, Group=, Trigger=doCow 8602, Actions=[EventTableActionDetach 8603], Comment=
EventTableTriggerIO 8602: Operator=0, IOValue=[0], IRC5Controller=? -1, SignalSource=SimulationProject 3637
EventTableActionDetach 8603: AttachmentParent=CowCatcherTool_R 5959, AttachmentChild=? -1
EventTableTriggerIO 8770: Operator=0, IOValue=[1], IRC5Controller=? -1, SignalSource=SimulationProject 3637
EventTableTriggerIO 8771: Operator=0, IOValue=[1], IRC5Controller=? -1, SignalSource=SimulationProject 3637
EventTableTriggerIO 8772: Operator=0, IOValue=[0], IRC5Controller=? -1, SignalSource=SimulationProject 3637
EventTableTriggerIO 8773: Operator=0, IOValue=[0], IRC5Controller=? -1, SignalSource=SimulationProject 3637
EventTableTriggerIO 8774: Operator=0, IOValue=[1], IRC5Controller=? -1, SignalSource=SimulationProject 3637
EventTableTriggerIO 8775: Operator=0, IOValue=[1], IRC5Controller=? -1, SignalSource=SimulationProject 3637
EventTableTriggerIO 8776: Operator=0, IOValue=[0], IRC5Controller=? -1, SignalSource=SimulationProject 3637
EventTableTriggerIO 8777: Operator=0, IOValue=[0], IRC5Controller=? -1, SignalSource=SimulationProject 3637
EventTableTriggerIO 8778: Operator=0, IOValue=[1], IRC5Controller=? -1, SignalSource=SimulationProject 3637
EventTableTriggerIO 8779: Operator=0, IOValue=[1], IRC5Controller=? -1, SignalSource=SimulationProject 3637
EventTableTriggerIO 8780: Operator=0, IOValue=[0], IRC5Controller=? -1, SignalSource=SimulationProject 3637
EventTableTriggerIO 8781: Operator=0, IOValue=[0], IRC5Controller=? -1, SignalSource=SimulationProject 3637
EventTableTriggerIO 8782: Operator=0, IOValue=[1], IRC5Controller=? -1, SignalSource=SimulationProject 3637
EventTableTriggerIO 8783: Operator=0, IOValue=[1], IRC5Controller=? -1, SignalSource=SimulationProject 3637
EventTableTriggerIO 8784: Operator=0, IOValue=[0], IRC5Controller=? -1, SignalSource=SimulationProject 3637
EventTableTriggerIO 8785: Operator=0, IOValue=[0], IRC5Controller=? -1, SignalSource=SimulationProject 3637
EventTableTriggerIO 8786: Operator=0, IOValue=[1], IRC5Controller=? -1, SignalSource=SimulationProject 3637
EventTableTriggerIO 8787: Operator=0, IOValue=[1], IRC5Controller=? -1, SignalSource=SimulationProject 3637
EventTableTriggerIO 8788: Operator=0, IOValue=[0], IRC5Controller=? -1, SignalSource=SimulationProject 3637
EventTableTriggerIO 8789: Operator=0, IOValue=[0], IRC5Controller=? -1, SignalSource=SimulationProject 3637
EventTableTriggerIO 8790: Operator=0, IOValue=[1], IRC5Controller=? -1, SignalSource=SimulationProject 3637
EventTableTriggerIO 8791: Operator=0, IOValue=[1], IRC5Controller=? -1, SignalSource=SimulationProject 3637
EventTableTriggerIO 8792: Operator=0, IOValue=[0], IRC5Controller=? -1, SignalSource=SimulationProject 3637
EventTableTriggerIO 8793: Operator=0, IOValue=[0], IRC5Controller=? -1, SignalSource=SimulationProject 3637
EventTableTriggerIO 8794: Operator=0, IOValue=[1], IRC5Controller=? -1, SignalSource=SimulationProject 3637
EventTableTriggerIO 8795: Operator=0, IOValue=[1], IRC5Controller=? -1, SignalSource=SimulationProject 3637
EventTableTriggerIO 8796: Operator=0, IOValue=[0], IRC5Controller=? -1, SignalSource=SimulationProject 3637
EventTableTriggerIO 8797: Operator=0, IOValue=[0], IRC5Controller=? -1, SignalSource=SimulationProject 3637
EventTableTriggerIO 8798: Operator=0, IOValue=[1], IRC5Controller=? -1, SignalSource=SimulationProject 3637
EventTableTriggerIO 8799: Operator=0, IOValue=[1], IRC5Controller=? -1, SignalSource=SimulationProject 3637
EventTableTriggerIO 8800: Operator=0, IOValue=[0], IRC5Controller=? -1, SignalSource=SimulationProject 3637
EventTableTriggerIO 8801: Operator=0, IOValue=[0], IRC5Controller=? -1, SignalSource=SimulationProject 3637
EventTableTriggerIO 8802: Operator=0, IOValue=[1], IRC5Controller=? -1, SignalSource=SimulationProject 3637
EventTableTriggerIO 8803: Operator=0, IOValue=[1], IRC5Controller=? -1, SignalSource=SimulationProject 3637
EventTableTriggerIO 8804: Operator=0, IOValue=[0], IRC5Controller=? -1, SignalSource=SimulationProject 3637
EventTableTriggerIO 8805: Operator=0, IOValue=[0], IRC5Controller=? -1, SignalSource=SimulationProject 3637
EventTableTriggerIO 8806: Operator=0, IOValue=[1], IRC5Controller=? -1, SignalSource=SimulationProject 3637
EventTableTriggerIO 8807: Operator=0, IOValue=[1], IRC5Controller=? -1, SignalSource=SimulationProject 3637
EventTableTriggerIO 8808: Operator=0, IOValue=[0], IRC5Controller=? -1, SignalSource=SimulationProject 3637
EventTableTriggerIO 8809: Operator=0, IOValue=[0], IRC5Controller=? -1, SignalSource=SimulationProject 3637
EventTableTriggerIO 8824: Operator=0, IOValue=[1], IRC5Controller=? -1, SignalSource=SimulationProject 3637
EventTableTriggerIO 8825: Operator=0, IOValue=[0], IRC5Controller=? -1, SignalSource=SimulationProject 3637
EventTableTriggerIO 8826: Operator=0, IOValue=[1], IRC5Controller=? -1, SignalSource=SimulationProject 3637
EventTableTriggerIO 8827: Operator=0, IOValue=[0], IRC5Controller=? -1, SignalSource=SimulationProject 3637
EventTableTriggerIO 8828: Operator=0, IOValue=[1], IRC5Controller=? -1, SignalSource=SimulationProject 3637
EventTableTriggerIO 8829: Operator=0, IOValue=[0], IRC5Controller=? -1, SignalSource=SimulationProject 3637
EventTableTriggerIO 8830: Operator=0, IOValue=[1], IRC5Controller=? -1, SignalSource=SimulationProject 3637
EventTableTriggerIO 8831: Operator=0, IOValue=[0], IRC5Controller=? -1, SignalSource=SimulationProject 3637
EventTableTriggerIO 8832: Operator=0, IOValue=[1], IRC5Controller=? -1, SignalSource=SimulationProject 3637
EventTableTriggerIO 8833: Operator=0, IOValue=[0], IRC5Controller=? -1, SignalSource=SimulationProject 3637
EventTableTriggerIO 8834: Operator=0, IOValue=[1], IRC5Controller=? -1, SignalSource=SimulationProject 3637
EventTableTriggerIO 8835: Operator=0, IOValue=[0], IRC5Controller=? -1, SignalSource=SimulationProject 3637
EventTableTriggerIO 8836: Operator=0, IOValue=[1], IRC5Controller=? -1, SignalSource=SimulationProject 3637
EventTableTriggerIO 8837: Operator=0, IOValue=[0], IRC5Controller=? -1, SignalSource=SimulationProject 3637
EventTableTriggerIO 8838: Operator=0, IOValue=[1], IRC5Controller=? -1, SignalSource=SimulationProject 3637
EventTableTriggerIO 8839: Operator=0, IOValue=[0], IRC5Controller=? -1, SignalSource=SimulationProject 3637
EventTableTriggerIO 8840: Operator=0, IOValue=[1], IRC5Controller=? -1, SignalSource=SimulationProject 3637
EventTableTriggerIO 8841: Operator=0, IOValue=[0], IRC5Controller=? -1, SignalSource=SimulationProject 3637
EventTableTriggerIO 8842: Operator=0, IOValue=[1], IRC5Controller=? -1, SignalSource=SimulationProject 3637
EventTableTriggerIO 8843: Operator=0, IOValue=[0], IRC5Controller=? -1, SignalSource=SimulationProject 3637
EventTableTriggerIO 8853: Operator=0, IOValue=[1], IRC5Controller=? -1, SignalSource=SimulationProject 3637
EventTableTriggerIO 8854: Operator=0, IOValue=[1], IRC5Controller=? -1, SignalSource=SimulationProject 3637
EventTableTriggerIO 8855: Operator=0, IOValue=[1], IRC5Controller=? -1, SignalSource=SimulationProject 3637
EventTableTriggerIO 8856: Operator=0, IOValue=[1], IRC5Controller=? -1, SignalSource=SimulationProject 3637
EventTableTriggerIO 8857: Operator=0, IOValue=[1], IRC5Controller=? -1, SignalSource=SimulationProject 3637
EventTableTriggerIO 8858: Operator=0, IOValue=[0], IRC5Controller=? -1, SignalSource=SimulationProject 3637
EventTableTriggerIO 8859: Operator=0, IOValue=[0], IRC5Controller=? -1, SignalSource=SimulationProject 3637
EventTableTriggerIO 8860: Operator=0, IOValue=[0], IRC5Controller=? -1, SignalSource=SimulationProject 3637
EventTableTriggerIO 8861: Operator=0, IOValue=[0], IRC5Controller=? -1, SignalSource=SimulationProject 3637
EventTableTriggerIO 8862: Operator=0, IOValue=[0], IRC5Controller=? -1, SignalSource=SimulationProject 3637
EventTableTriggerIO 8863: Operator=0, IOValue=[1], IRC5Controller=? -1, SignalSource=SimulationProject 3637
EventTableTriggerIO 8864: Operator=0, IOValue=[1], IRC5Controller=? -1, SignalSource=SimulationProject 3637
EventTableTriggerIO 8865: Operator=0, IOValue=[1], IRC5Controller=? -1, SignalSource=SimulationProject 3637
EventTableTriggerIO 8866: Operator=0, IOValue=[1], IRC5Controller=? -1, SignalSource=SimulationProject 3637
EventTableTriggerIO 8867: Operator=0, IOValue=[1], IRC5Controller=? -1, SignalSource=SimulationProject 3637
EventTableTriggerIO 8868: Operator=0, IOValue=[0], IRC5Controller=? -1, SignalSource=SimulationProject 3637
EventTableTriggerIO 8869: Operator=0, IOValue=[0], IRC5Controller=? -1, SignalSource=SimulationProject 3637
EventTableTriggerIO 8870: Operator=0, IOValue=[0], IRC5Controller=? -1, SignalSource=SimulationProject 3637
EventTableTriggerIO 8871: Operator=0, IOValue=[0], IRC5Controller=? -1, SignalSource=SimulationProject 3637
EventTableTriggerIO 8872: Operator=0, IOValue=[0], IRC5Controller=? -1, SignalSource=SimulationProject 3637
EventTableTriggerIO 8873: Operator=0, IOValue=[1], IRC5Controller=? -1, SignalSource=SimulationProject 3637
EventTableTriggerIO 8874: Operator=0, IOValue=[1], IRC5Controller=? -1, SignalSource=SimulationProject 3637
EventTableTriggerIO 8875: Operator=0, IOValue=[1], IRC5Controller=? -1, SignalSource=SimulationProject 3637
EventTableTriggerIO 8876: Operator=0, IOValue=[1], IRC5Controller=? -1, SignalSource=SimulationProject 3637
EventTableTriggerIO 8877: Operator=0, IOValue=[1], IRC5Controller=? -1, SignalSource=SimulationProject 3637
EventTableTriggerIO 8878: Operator=0, IOValue=[0], IRC5Controller=? -1, SignalSource=SimulationProject 3637
EventTableTriggerIO 8879: Operator=0, IOValue=[0], IRC5Controller=? -1, SignalSource=SimulationProject 3637
EventTableTriggerIO 8880: Operator=0, IOValue=[0], IRC5Controller=? -1, SignalSource=SimulationProject 3637
EventTableTriggerIO 8881: Operator=0, IOValue=[0], IRC5Controller=? -1, SignalSource=SimulationProject 3637
EventTableTriggerIO 8882: Operator=0, IOValue=[0], IRC5Controller=? -1, SignalSource=SimulationProject 3637
EventTableTriggerIO 8883: Operator=0, IOValue=[1], IRC5Controller=? -1, SignalSource=SimulationProject 3637
EventTableTriggerIO 8884: Operator=0, IOValue=[1], IRC5Controller=? -1, SignalSource=SimulationProject 3637
EventTableTriggerIO 8885: Operator=0, IOValue=[1], IRC5Controller=? -1, SignalSource=SimulationProject 3637
EventTableTriggerIO 8886: Operator=0, IOValue=[1], IRC5Controller=? -1, SignalSource=SimulationProject 3637
EventTableTriggerIO 8887: Operator=0, IOValue=[1], IRC5Controller=? -1, SignalSource=SimulationProject 3637
EventTableTriggerIO 8888: Operator=0, IOValue=[0], IRC5Controller=? -1, SignalSource=SimulationProject 3637
EventTableTriggerIO 8889: Operator=0, IOValue=[0], IRC5Controller=? -1, SignalSource=SimulationProject 3637
EventTableTriggerIO 8890: Operator=0, IOValue=[0], IRC5Controller=? -1, SignalSource=SimulationProject 3637
EventTableTriggerIO 8891: Operator=0, IOValue=[0], IRC5Controller=? -1, SignalSource=SimulationProject 3637
EventTableTriggerIO 8892: Operator=0, IOValue=[0], IRC5Controller=? -1, SignalSource=SimulationProject 3637
EventTableTriggerIO 8893: Operator=0, IOValue=[1], IRC5Controller=? -1, SignalSource=SimulationProject 3637
EventTableTriggerIO 8894: Operator=0, IOValue=[1], IRC5Controller=? -1, SignalSource=SimulationProject 3637
EventTableTriggerIO 8895: Operator=0, IOValue=[1], IRC5Controller=? -1, SignalSource=SimulationProject 3637
EventTableTriggerIO 8896: Operator=0, IOValue=[1], IRC5Controller=? -1, SignalSource=SimulationProject 3637
EventTableTriggerIO 8897: Operator=0, IOValue=[1], IRC5Controller=? -1, SignalSource=SimulationProject 3637
EventTableTriggerIO 8898: Operator=0, IOValue=[0], IRC5Controller=? -1, SignalSource=SimulationProject 3637
EventTableTriggerIO 8899: Operator=0, IOValue=[0], IRC5Controller=? -1, SignalSource=SimulationProject 3637
EventTableTriggerIO 8900: Operator=0, IOValue=[0], IRC5Controller=? -1, SignalSource=SimulationProject 3637
EventTableTriggerIO 8901: Operator=0, IOValue=[0], IRC5Controller=? -1, SignalSource=SimulationProject 3637
EventTableTriggerIO 8902: Operator=0, IOValue=[0], IRC5Controller=? -1, SignalSource=SimulationProject 3637
EventTableTriggerIO 8903: Operator=0, IOValue=[1], IRC5Controller=? -1, SignalSource=SimulationProject 3637
EventTableTriggerIO 8904: Operator=0, IOValue=[1], IRC5Controller=? -1, SignalSource=SimulationProject 3637
EventTableTriggerIO 8905: Operator=0, IOValue=[1], IRC5Controller=? -1, SignalSource=SimulationProject 3637
EventTableTriggerIO 8906: Operator=0, IOValue=[1], IRC5Controller=? -1, SignalSource=SimulationProject 3637
EventTableTriggerIO 8907: Operator=0, IOValue=[1], IRC5Controller=? -1, SignalSource=SimulationProject 3637
EventTableTriggerIO 8908: Operator=0, IOValue=[0], IRC5Controller=? -1, SignalSource=SimulationProject 3637
EventTableTriggerIO 8909: Operator=0, IOValue=[0], IRC5Controller=? -1, SignalSource=SimulationProject 3637
EventTableTriggerIO 8910: Operator=0, IOValue=[0], IRC5Controller=? -1, SignalSource=SimulationProject 3637
EventTableTriggerIO 8911: Operator=0, IOValue=[0], IRC5Controller=? -1, SignalSource=SimulationProject 3637
EventTableTriggerIO 8912: Operator=0, IOValue=[0], IRC5Controller=? -1, SignalSource=SimulationProject 3637
EventTableTriggerIO 8913: Operator=0, IOValue=[1], IRC5Controller=? -1, SignalSource=SimulationProject 3637
EventTableTriggerIO 8914: Operator=0, IOValue=[1], IRC5Controller=? -1, SignalSource=SimulationProject 3637
EventTableTriggerIO 8915: Operator=0, IOValue=[1], IRC5Controller=? -1, SignalSource=SimulationProject 3637
EventTableTriggerIO 8916: Operator=0, IOValue=[1], IRC5Controller=? -1, SignalSource=SimulationProject 3637
EventTableTriggerIO 8917: Operator=0, IOValue=[1], IRC5Controller=? -1, SignalSource=SimulationProject 3637
EventTableTriggerIO 8918: Operator=0, IOValue=[0], IRC5Controller=? -1, SignalSource=SimulationProject 3637
EventTableTriggerIO 8919: Operator=0, IOValue=[0], IRC5Controller=? -1, SignalSource=SimulationProject 3637
EventTableTriggerIO 8920: Operator=0, IOValue=[0], IRC5Controller=? -1, SignalSource=SimulationProject 3637
EventTableTriggerIO 8921: Operator=0, IOValue=[0], IRC5Controller=? -1, SignalSource=SimulationProject 3637
EventTableTriggerIO 8922: Operator=0, IOValue=[0], IRC5Controller=? -1, SignalSource=SimulationProject 3637
EventTableTriggerIO 8923: Operator=0, IOValue=[1], IRC5Controller=? -1, SignalSource=SimulationProject 3637
EventTableTriggerIO 8924: Operator=0, IOValue=[1], IRC5Controller=? -1, SignalSource=SimulationProject 3637
EventTableTriggerIO 8925: Operator=0, IOValue=[1], IRC5Controller=? -1, SignalSource=SimulationProject 3637
EventTableTriggerIO 8926: Operator=0, IOValue=[1], IRC5Controller=? -1, SignalSource=SimulationProject 3637
EventTableTriggerIO 8927: Operator=0, IOValue=[1], IRC5Controller=? -1, SignalSource=SimulationProject 3637
EventTableTriggerIO 8928: Operator=0, IOValue=[0], IRC5Controller=? -1, SignalSource=SimulationProject 3637
EventTableTriggerIO 8929: Operator=0, IOValue=[0], IRC5Controller=? -1, SignalSource=SimulationProject 3637
EventTableTriggerIO 8930: Operator=0, IOValue=[0], IRC5Controller=? -1, SignalSource=SimulationProject 3637
EventTableTriggerIO 8931: Operator=0, IOValue=[0], IRC5Controller=? -1, SignalSource=SimulationProject 3637
EventTableTriggerIO 8932: Operator=0, IOValue=[0], IRC5Controller=? -1, SignalSource=SimulationProject 3637
EventTableTriggerIO 8933: Operator=0, IOValue=[1], IRC5Controller=? -1, SignalSource=SimulationProject 3637
EventTableTriggerIO 8934: Operator=0, IOValue=[1], IRC5Controller=? -1, SignalSource=SimulationProject 3637
EventTableTriggerIO 8935: Operator=0, IOValue=[1], IRC5Controller=? -1, SignalSource=SimulationProject 3637
EventTableTriggerIO 8936: Operator=0, IOValue=[1], IRC5Controller=? -1, SignalSource=SimulationProject 3637
EventTableTriggerIO 8937: Operator=0, IOValue=[1], IRC5Controller=? -1, SignalSource=SimulationProject 3637
EventTableTriggerIO 8938: Operator=0, IOValue=[0], IRC5Controller=? -1, SignalSource=SimulationProject 3637
EventTableTriggerIO 8939: Operator=0, IOValue=[0], IRC5Controller=? -1, SignalSource=SimulationProject 3637
EventTableTriggerIO 8940: Operator=0, IOValue=[0], IRC5Controller=? -1, SignalSource=SimulationProject 3637
EventTableTriggerIO 8941: Operator=0, IOValue=[0], IRC5Controller=? -1, SignalSource=SimulationProject 3637
EventTableTriggerIO 8942: Operator=0, IOValue=[0], IRC5Controller=? -1, SignalSource=SimulationProject 3637
EventTableTriggerIO 8943: Operator=0, IOValue=[1], IRC5Controller=? -1, SignalSource=SimulationProject 3637
EventTableTriggerIO 8944: Operator=0, IOValue=[1], IRC5Controller=? -1, SignalSource=SimulationProject 3637
EventTableTriggerIO 8945: Operator=0, IOValue=[1], IRC5Controller=? -1, SignalSource=SimulationProject 3637
EventTableTriggerIO 8946: Operator=0, IOValue=[1], IRC5Controller=? -1, SignalSource=SimulationProject 3637
EventTableTriggerIO 8947: Operator=0, IOValue=[1], IRC5Controller=? -1, SignalSource=SimulationProject 3637
EventTableTriggerIO 8948: Operator=0, IOValue=[0], IRC5Controller=? -1, SignalSource=SimulationProject 3637
EventTableTriggerIO 8949: Operator=0, IOValue=[0], IRC5Controller=? -1, SignalSource=SimulationProject 3637
EventTableTriggerIO 8950: Operator=0, IOValue=[0], IRC5Controller=? -1, SignalSource=SimulationProject 3637
EventTableTriggerIO 8951: Operator=0, IOValue=[0], IRC5Controller=? -1, SignalSource=SimulationProject 3637
EventTableTriggerIO 8952: Operator=0, IOValue=[0], IRC5Controller=? -1, SignalSource=SimulationProject 3637
EventTableTriggerIO 8981: Operator=0, IOValue=[1], IRC5Controller=? -1, SignalSource=SimulationProject 3637
EventTableTriggerIO 8982: Operator=0, IOValue=[1], IRC5Controller=? -1, SignalSource=SimulationProject 3637
EventTableTriggerIO 8983: Operator=0, IOValue=[1], IRC5Controller=? -1, SignalSource=SimulationProject 3637
EventTableTriggerIO 8984: Operator=0, IOValue=[1], IRC5Controller=? -1, SignalSource=SimulationProject 3637
EventTableTriggerIO 8985: Operator=0, IOValue=[0], IRC5Controller=? -1, SignalSource=SimulationProject 3637
EventTableTriggerIO 8986: Operator=0, IOValue=[0], IRC5Controller=? -1, SignalSource=SimulationProject 3637
EventTableTriggerIO 8987: Operator=0, IOValue=[0], IRC5Controller=? -1, SignalSource=SimulationProject 3637
EventTableTriggerIO 8988: Operator=0, IOValue=[0], IRC5Controller=? -1, SignalSource=SimulationProject 3637
EventTableTriggerIO 8989: Operator=0, IOValue=[1], IRC5Controller=? -1, SignalSource=SimulationProject 3637
EventTableTriggerIO 8990: Operator=0, IOValue=[1], IRC5Controller=? -1, SignalSource=SimulationProject 3637
EventTableTriggerIO 8991: Operator=0, IOValue=[1], IRC5Controller=? -1, SignalSource=SimulationProject 3637
EventTableTriggerIO 8992: Operator=0, IOValue=[1], IRC5Controller=? -1, SignalSource=SimulationProject 3637
EventTableTriggerIO 8993: Operator=0, IOValue=[0], IRC5Controller=? -1, SignalSource=SimulationProject 3637
EventTableTriggerIO 8994: Operator=0, IOValue=[0], IRC5Controller=? -1, SignalSource=SimulationProject 3637
EventTableTriggerIO 8995: Operator=0, IOValue=[0], IRC5Controller=? -1, SignalSource=SimulationProject 3637
EventTableTriggerIO 8996: Operator=0, IOValue=[0], IRC5Controller=? -1, SignalSource=SimulationProject 3637
EventTableTriggerIO 8997: Operator=0, IOValue=[1], IRC5Controller=? -1, SignalSource=SimulationProject 3637
EventTableTriggerIO 8998: Operator=0, IOValue=[1], IRC5Controller=? -1, SignalSource=SimulationProject 3637
EventTableTriggerIO 8999: Operator=0, IOValue=[1], IRC5Controller=? -1, SignalSource=SimulationProject 3637
EventTableTriggerIO 9000: Operator=0, IOValue=[1], IRC5Controller=? -1, SignalSource=SimulationProject 3637
EventTableTriggerIO 9001: Operator=0, IOValue=[0], IRC5Controller=? -1, SignalSource=SimulationProject 3637
EventTableTriggerIO 9002: Operator=0, IOValue=[0], IRC5Controller=? -1, SignalSource=SimulationProject 3637
EventTableTriggerIO 9003: Operator=0, IOValue=[0], IRC5Controller=? -1, SignalSource=SimulationProject 3637
EventTableTriggerIO 9004: Operator=0, IOValue=[0], IRC5Controller=? -1, SignalSource=SimulationProject 3637
EventTableTriggerIO 9005: Operator=0, IOValue=[1], IRC5Controller=? -1, SignalSource=SimulationProject 3637
EventTableTriggerIO 9006: Operator=0, IOValue=[1], IRC5Controller=? -1, SignalSource=SimulationProject 3637
EventTableTriggerIO 9007: Operator=0, IOValue=[1], IRC5Controller=? -1, SignalSource=SimulationProject 3637
EventTableTriggerIO 9008: Operator=0, IOValue=[1], IRC5Controller=? -1, SignalSource=SimulationProject 3637
EventTableTriggerIO 9009: Operator=0, IOValue=[0], IRC5Controller=? -1, SignalSource=SimulationProject 3637
EventTableTriggerIO 9010: Operator=0, IOValue=[0], IRC5Controller=? -1, SignalSource=SimulationProject 3637
EventTableTriggerIO 9011: Operator=0, IOValue=[0], IRC5Controller=? -1, SignalSource=SimulationProject 3637
EventTableTriggerIO 9012: Operator=0, IOValue=[0], IRC5Controller=? -1, SignalSource=SimulationProject 3637
EventTableTriggerIO 9013: Operator=0, IOValue=[1], IRC5Controller=? -1, SignalSource=SimulationProject 3637
EventTableTriggerIO 9014: Operator=0, IOValue=[1], IRC5Controller=? -1, SignalSource=SimulationProject 3637
EventTableTriggerIO 9015: Operator=0, IOValue=[1], IRC5Controller=? -1, SignalSource=SimulationProject 3637
EventTableTriggerIO 9016: Operator=0, IOValue=[1], IRC5Controller=? -1, SignalSource=SimulationProject 3637
EventTableTriggerIO 9017: Operator=0, IOValue=[0], IRC5Controller=? -1, SignalSource=SimulationProject 3637
EventTableTriggerIO 9018: Operator=0, IOValue=[0], IRC5Controller=? -1, SignalSource=SimulationProject 3637
EventTableTriggerIO 9019: Operator=0, IOValue=[0], IRC5Controller=? -1, SignalSource=SimulationProject 3637
EventTableTriggerIO 9020: Operator=0, IOValue=[0], IRC5Controller=? -1, SignalSource=SimulationProject 3637
EventTableTriggerIO 9021: Operator=0, IOValue=[1], IRC5Controller=? -1, SignalSource=SimulationProject 3637
EventTableTriggerIO 9022: Operator=0, IOValue=[1], IRC5Controller=? -1, SignalSource=SimulationProject 3637
EventTableTriggerIO 9023: Operator=0, IOValue=[1], IRC5Controller=? -1, SignalSource=SimulationProject 3637
EventTableTriggerIO 9024: Operator=0, IOValue=[1], IRC5Controller=? -1, SignalSource=SimulationProject 3637
EventTableTriggerIO 9025: Operator=0, IOValue=[0], IRC5Controller=? -1, SignalSource=SimulationProject 3637
EventTableTriggerIO 9026: Operator=0, IOValue=[0], IRC5Controller=? -1, SignalSource=SimulationProject 3637
EventTableTriggerIO 9027: Operator=0, IOValue=[0], IRC5Controller=? -1, SignalSource=SimulationProject 3637
EventTableTriggerIO 9028: Operator=0, IOValue=[0], IRC5Controller=? -1, SignalSource=SimulationProject 3637
EventTableTriggerIO 9029: Operator=0, IOValue=[1], IRC5Controller=? -1, SignalSource=SimulationProject 3637
EventTableTriggerIO 9030: Operator=0, IOValue=[1], IRC5Controller=? -1, SignalSource=SimulationProject 3637
EventTableTriggerIO 9031: Operator=0, IOValue=[1], IRC5Controller=? -1, SignalSource=SimulationProject 3637
EventTableTriggerIO 9032: Operator=0, IOValue=[1], IRC5Controller=? -1, SignalSource=SimulationProject 3637
EventTableTriggerIO 9033: Operator=0, IOValue=[0], IRC5Controller=? -1, SignalSource=SimulationProject 3637
EventTableTriggerIO 9034: Operator=0, IOValue=[0], IRC5Controller=? -1, SignalSource=SimulationProject 3637
EventTableTriggerIO 9035: Operator=0, IOValue=[0], IRC5Controller=? -1, SignalSource=SimulationProject 3637
EventTableTriggerIO 9036: Operator=0, IOValue=[0], IRC5Controller=? -1, SignalSource=SimulationProject 3637
EventTableTriggerIO 9037: Operator=0, IOValue=[1], IRC5Controller=? -1, SignalSource=SimulationProject 3637
EventTableTriggerIO 9038: Operator=0, IOValue=[1], IRC5Controller=? -1, SignalSource=SimulationProject 3637
EventTableTriggerIO 9039: Operator=0, IOValue=[1], IRC5Controller=? -1, SignalSource=SimulationProject 3637
EventTableTriggerIO 9040: Operator=0, IOValue=[1], IRC5Controller=? -1, SignalSource=SimulationProject 3637
EventTableTriggerIO 9041: Operator=0, IOValue=[0], IRC5Controller=? -1, SignalSource=SimulationProject 3637
EventTableTriggerIO 9042: Operator=0, IOValue=[0], IRC5Controller=? -1, SignalSource=SimulationProject 3637
EventTableTriggerIO 9043: Operator=0, IOValue=[0], IRC5Controller=? -1, SignalSource=SimulationProject 3637
EventTableTriggerIO 9044: Operator=0, IOValue=[0], IRC5Controller=? -1, SignalSource=SimulationProject 3637
EventTableTriggerIO 9045: Operator=0, IOValue=[1], IRC5Controller=? -1, SignalSource=SimulationProject 3637
EventTableTriggerIO 9046: Operator=0, IOValue=[1], IRC5Controller=? -1, SignalSource=SimulationProject 3637
EventTableTriggerIO 9047: Operator=0, IOValue=[1], IRC5Controller=? -1, SignalSource=SimulationProject 3637
EventTableTriggerIO 9048: Operator=0, IOValue=[1], IRC5Controller=? -1, SignalSource=SimulationProject 3637
EventTableTriggerIO 9049: Operator=0, IOValue=[0], IRC5Controller=? -1, SignalSource=SimulationProject 3637
EventTableTriggerIO 9050: Operator=0, IOValue=[0], IRC5Controller=? -1, SignalSource=SimulationProject 3637
EventTableTriggerIO 9051: Operator=0, IOValue=[0], IRC5Controller=? -1, SignalSource=SimulationProject 3637
EventTableTriggerIO 9052: Operator=0, IOValue=[0], IRC5Controller=? -1, SignalSource=SimulationProject 3637
EventTableTriggerIO 9053: Operator=0, IOValue=[1], IRC5Controller=? -1, SignalSource=SimulationProject 3637
EventTableTriggerIO 9054: Operator=0, IOValue=[1], IRC5Controller=? -1, SignalSource=SimulationProject 3637
EventTableTriggerIO 9055: Operator=0, IOValue=[1], IRC5Controller=? -1, SignalSource=SimulationProject 3637
EventTableTriggerIO 9056: Operator=0, IOValue=[1], IRC5Controller=? -1, SignalSource=SimulationProject 3637
EventTableTriggerIO 9057: Operator=0, IOValue=[0], IRC5Controller=? -1, SignalSource=SimulationProject 3637
EventTableTriggerIO 9058: Operator=0, IOValue=[0], IRC5Controller=? -1, SignalSource=SimulationProject 3637
EventTableTriggerIO 9059: Operator=0, IOValue=[0], IRC5Controller=? -1, SignalSource=SimulationProject 3637
EventTableTriggerIO 9060: Operator=0, IOValue=[0], IRC5Controller=? -1, SignalSource=SimulationProject 3637
EventTableTriggerIO 9075: Operator=0, IOValue=[1], IRC5Controller=? -1, SignalSource=SimulationProject 3637
EventTableTriggerIO 9076: Operator=0, IOValue=[1], IRC5Controller=? -1, SignalSource=SimulationProject 3637
EventTableTriggerIO 9077: Operator=0, IOValue=[1], IRC5Controller=? -1, SignalSource=SimulationProject 3637
EventTableTriggerIO 9078: Operator=0, IOValue=[1], IRC5Controller=? -1, SignalSource=SimulationProject 3637
EventTableTriggerIO 9079: Operator=0, IOValue=[1], IRC5Controller=? -1, SignalSource=SimulationProject 3637
EventTableTriggerIO 9080: Operator=0, IOValue=[1], IRC5Controller=? -1, SignalSource=SimulationProject 3637
EventTableTriggerIO 9081: Operator=0, IOValue=[1], IRC5Controller=? -1, SignalSource=SimulationProject 3637
EventTableTriggerIO 9082: Operator=0, IOValue=[0], IRC5Controller=? -1, SignalSource=SimulationProject 3637
EventTableTriggerIO 9083: Operator=0, IOValue=[0], IRC5Controller=? -1, SignalSource=SimulationProject 3637
EventTableTriggerIO 9084: Operator=0, IOValue=[0], IRC5Controller=? -1, SignalSource=SimulationProject 3637
EventTableTriggerIO 9085: Operator=0, IOValue=[0], IRC5Controller=? -1, SignalSource=SimulationProject 3637
EventTableTriggerIO 9086: Operator=0, IOValue=[0], IRC5Controller=? -1, SignalSource=SimulationProject 3637
EventTableTriggerIO 9087: Operator=0, IOValue=[0], IRC5Controller=? -1, SignalSource=SimulationProject 3637
EventTableTriggerIO 9088: Operator=0, IOValue=[0], IRC5Controller=? -1, SignalSource=SimulationProject 3637
EventTableTriggerIO 9089: Operator=0, IOValue=[1], IRC5Controller=? -1, SignalSource=SimulationProject 3637
EventTableTriggerIO 9090: Operator=0, IOValue=[1], IRC5Controller=? -1, SignalSource=SimulationProject 3637
EventTableTriggerIO 9091: Operator=0, IOValue=[1], IRC5Controller=? -1, SignalSource=SimulationProject 3637
EventTableTriggerIO 9092: Operator=0, IOValue=[1], IRC5Controller=? -1, SignalSource=SimulationProject 3637
EventTableTriggerIO 9093: Operator=0, IOValue=[1], IRC5Controller=? -1, SignalSource=SimulationProject 3637
EventTableTriggerIO 9094: Operator=0, IOValue=[1], IRC5Controller=? -1, SignalSource=SimulationProject 3637
EventTableTriggerIO 9095: Operator=0, IOValue=[1], IRC5Controller=? -1, SignalSource=SimulationProject 3637
EventTableTriggerIO 9096: Operator=0, IOValue=[0], IRC5Controller=? -1, SignalSource=SimulationProject 3637
EventTableTriggerIO 9097: Operator=0, IOValue=[0], IRC5Controller=? -1, SignalSource=SimulationProject 3637
EventTableTriggerIO 9098: Operator=0, IOValue=[0], IRC5Controller=? -1, SignalSource=SimulationProject 3637
EventTableTriggerIO 9099: Operator=0, IOValue=[0], IRC5Controller=? -1, SignalSource=SimulationProject 3637
EventTableTriggerIO 9100: Operator=0, IOValue=[0], IRC5Controller=? -1, SignalSource=SimulationProject 3637
EventTableTriggerIO 9101: Operator=0, IOValue=[0], IRC5Controller=? -1, SignalSource=SimulationProject 3637
EventTableTriggerIO 9102: Operator=0, IOValue=[0], IRC5Controller=? -1, SignalSource=SimulationProject 3637
EventTableTriggerIO 9103: Operator=0, IOValue=[1], IRC5Controller=? -1, SignalSource=SimulationProject 3637
EventTableTriggerIO 9104: Operator=0, IOValue=[1], IRC5Controller=? -1, SignalSource=SimulationProject 3637
EventTableTriggerIO 9105: Operator=0, IOValue=[1], IRC5Controller=? -1, SignalSource=SimulationProject 3637
EventTableTriggerIO 9106: Operator=0, IOValue=[1], IRC5Controller=? -1, SignalSource=SimulationProject 3637
EventTableTriggerIO 9107: Operator=0, IOValue=[1], IRC5Controller=? -1, SignalSource=SimulationProject 3637
EventTableTriggerIO 9108: Operator=0, IOValue=[1], IRC5Controller=? -1, SignalSource=SimulationProject 3637
EventTableTriggerIO 9109: Operator=0, IOValue=[1], IRC5Controller=? -1, SignalSource=SimulationProject 3637
EventTableTriggerIO 9110: Operator=0, IOValue=[0], IRC5Controller=? -1, SignalSource=SimulationProject 3637
EventTableTriggerIO 9111: Operator=0, IOValue=[0], IRC5Controller=? -1, SignalSource=SimulationProject 3637
EventTableTriggerIO 9112: Operator=0, IOValue=[0], IRC5Controller=? -1, SignalSource=SimulationProject 3637
EventTableTriggerIO 9113: Operator=0, IOValue=[0], IRC5Controller=? -1, SignalSource=SimulationProject 3637
EventTableTriggerIO 9114: Operator=0, IOValue=[0], IRC5Controller=? -1, SignalSource=SimulationProject 3637
EventTableTriggerIO 9115: Operator=0, IOValue=[0], IRC5Controller=? -1, SignalSource=SimulationProject 3637
EventTableTriggerIO 9116: Operator=0, IOValue=[0], IRC5Controller=? -1, SignalSource=SimulationProject 3637
EventTableTriggerIO 9117: Operator=0, IOValue=[1], IRC5Controller=? -1, SignalSource=SimulationProject 3637
EventTableTriggerIO 9118: Operator=0, IOValue=[1], IRC5Controller=? -1, SignalSource=SimulationProject 3637
EventTableTriggerIO 9119: Operator=0, IOValue=[1], IRC5Controller=? -1, SignalSource=SimulationProject 3637
EventTableTriggerIO 9120: Operator=0, IOValue=[1], IRC5Controller=? -1, SignalSource=SimulationProject 3637
EventTableTriggerIO 9121: Operator=0, IOValue=[1], IRC5Controller=? -1, SignalSource=SimulationProject 3637
EventTableTriggerIO 9122: Operator=0, IOValue=[1], IRC5Controller=? -1, SignalSource=SimulationProject 3637
EventTableTriggerIO 9123: Operator=0, IOValue=[1], IRC5Controller=? -1, SignalSource=SimulationProject 3637
EventTableTriggerIO 9124: Operator=0, IOValue=[0], IRC5Controller=? -1, SignalSource=SimulationProject 3637
EventTableTriggerIO 9125: Operator=0, IOValue=[0], IRC5Controller=? -1, SignalSource=SimulationProject 3637
EventTableTriggerIO 9126: Operator=0, IOValue=[0], IRC5Controller=? -1, SignalSource=SimulationProject 3637
EventTableTriggerIO 9127: Operator=0, IOValue=[0], IRC5Controller=? -1, SignalSource=SimulationProject 3637
EventTableTriggerIO 9128: Operator=0, IOValue=[0], IRC5Controller=? -1, SignalSource=SimulationProject 3637
EventTableTriggerIO 9129: Operator=0, IOValue=[0], IRC5Controller=? -1, SignalSource=SimulationProject 3637
EventTableTriggerIO 9130: Operator=0, IOValue=[0], IRC5Controller=? -1, SignalSource=SimulationProject 3637
EventTableTriggerIO 9131: Operator=0, IOValue=[1], IRC5Controller=? -1, SignalSource=SimulationProject 3637
EventTableTriggerIO 9132: Operator=0, IOValue=[1], IRC5Controller=? -1, SignalSource=SimulationProject 3637
EventTableTriggerIO 9133: Operator=0, IOValue=[1], IRC5Controller=? -1, SignalSource=SimulationProject 3637
EventTableTriggerIO 9134: Operator=0, IOValue=[1], IRC5Controller=? -1, SignalSource=SimulationProject 3637
EventTableTriggerIO 9135: Operator=0, IOValue=[1], IRC5Controller=? -1, SignalSource=SimulationProject 3637
EventTableTriggerIO 9136: Operator=0, IOValue=[1], IRC5Controller=? -1, SignalSource=SimulationProject 3637
EventTableTriggerIO 9137: Operator=0, IOValue=[1], IRC5Controller=? -1, SignalSource=SimulationProject 3637
EventTableTriggerIO 9138: Operator=0, IOValue=[0], IRC5Controller=? -1, SignalSource=SimulationProject 3637
EventTableTriggerIO 9139: Operator=0, IOValue=[0], IRC5Controller=? -1, SignalSource=SimulationProject 3637
EventTableTriggerIO 9140: Operator=0, IOValue=[0], IRC5Controller=? -1, SignalSource=SimulationProject 3637
EventTableTriggerIO 9141: Operator=0, IOValue=[0], IRC5Controller=? -1, SignalSource=SimulationProject 3637
EventTableTriggerIO 9142: Operator=0, IOValue=[0], IRC5Controller=? -1, SignalSource=SimulationProject 3637
EventTableTriggerIO 9143: Operator=0, IOValue=[0], IRC5Controller=? -1, SignalSource=SimulationProject 3637
EventTableTriggerIO 9144: Operator=0, IOValue=[0], IRC5Controller=? -1, SignalSource=SimulationProject 3637
EventTableTriggerIO 9145: Operator=0, IOValue=[1], IRC5Controller=? -1, SignalSource=SimulationProject 3637
EventTableTriggerIO 9146: Operator=0, IOValue=[1], IRC5Controller=? -1, SignalSource=SimulationProject 3637
EventTableTriggerIO 9147: Operator=0, IOValue=[1], IRC5Controller=? -1, SignalSource=SimulationProject 3637
EventTableTriggerIO 9148: Operator=0, IOValue=[1], IRC5Controller=? -1, SignalSource=SimulationProject 3637
EventTableTriggerIO 9149: Operator=0, IOValue=[1], IRC5Controller=? -1, SignalSource=SimulationProject 3637
EventTableTriggerIO 9150: Operator=0, IOValue=[1], IRC5Controller=? -1, SignalSource=SimulationProject 3637
EventTableTriggerIO 9151: Operator=0, IOValue=[1], IRC5Controller=? -1, SignalSource=SimulationProject 3637
EventTableTriggerIO 9152: Operator=0, IOValue=[0], IRC5Controller=? -1, SignalSource=SimulationProject 3637
EventTableTriggerIO 9153: Operator=0, IOValue=[0], IRC5Controller=? -1, SignalSource=SimulationProject 3637
EventTableTriggerIO 9154: Operator=0, IOValue=[0], IRC5Controller=? -1, SignalSource=SimulationProject 3637
EventTableTriggerIO 9155: Operator=0, IOValue=[0], IRC5Controller=? -1, SignalSource=SimulationProject 3637
EventTableTriggerIO 9156: Operator=0, IOValue=[0], IRC5Controller=? -1, SignalSource=SimulationProject 3637
EventTableTriggerIO 9157: Operator=0, IOValue=[0], IRC5Controller=? -1, SignalSource=SimulationProject 3637
EventTableTriggerIO 9158: Operator=0, IOValue=[0], IRC5Controller=? -1, SignalSource=SimulationProject 3637
EventTableTriggerIO 9159: Operator=0, IOValue=[1], IRC5Controller=? -1, SignalSource=SimulationProject 3637
EventTableTriggerIO 9160: Operator=0, IOValue=[1], IRC5Controller=? -1, SignalSource=SimulationProject 3637
EventTableTriggerIO 9161: Operator=0, IOValue=[1], IRC5Controller=? -1, SignalSource=SimulationProject 3637
EventTableTriggerIO 9162: Operator=0, IOValue=[1], IRC5Controller=? -1, SignalSource=SimulationProject 3637
EventTableTriggerIO 9163: Operator=0, IOValue=[1], IRC5Controller=? -1, SignalSource=SimulationProject 3637
EventTableTriggerIO 9164: Operator=0, IOValue=[1], IRC5Controller=? -1, SignalSource=SimulationProject 3637
EventTableTriggerIO 9165: Operator=0, IOValue=[1], IRC5Controller=? -1, SignalSource=SimulationProject 3637
EventTableTriggerIO 9166: Operator=0, IOValue=[0], IRC5Controller=? -1, SignalSource=SimulationProject 3637
EventTableTriggerIO 9167: Operator=0, IOValue=[0], IRC5Controller=? -1, SignalSource=SimulationProject 3637
EventTableTriggerIO 9168: Operator=0, IOValue=[0], IRC5Controller=? -1, SignalSource=SimulationProject 3637
EventTableTriggerIO 9169: Operator=0, IOValue=[0], IRC5Controller=? -1, SignalSource=SimulationProject 3637
EventTableTriggerIO 9170: Operator=0, IOValue=[0], IRC5Controller=? -1, SignalSource=SimulationProject 3637
EventTableTriggerIO 9171: Operator=0, IOValue=[0], IRC5Controller=? -1, SignalSource=SimulationProject 3637
EventTableTriggerIO 9172: Operator=0, IOValue=[0], IRC5Controller=? -1, SignalSource=SimulationProject 3637
EventTableTriggerIO 9173: Operator=0, IOValue=[1], IRC5Controller=? -1, SignalSource=SimulationProject 3637
EventTableTriggerIO 9174: Operator=0, IOValue=[1], IRC5Controller=? -1, SignalSource=SimulationProject 3637
EventTableTriggerIO 9175: Operator=0, IOValue=[1], IRC5Controller=? -1, SignalSource=SimulationProject 3637
EventTableTriggerIO 9176: Operator=0, IOValue=[1], IRC5Controller=? -1, SignalSource=SimulationProject 3637
EventTableTriggerIO 9177: Operator=0, IOValue=[1], IRC5Controller=? -1, SignalSource=SimulationProject 3637
EventTableTriggerIO 9178: Operator=0, IOValue=[1], IRC5Controller=? -1, SignalSource=SimulationProject 3637
EventTableTriggerIO 9179: Operator=0, IOValue=[1], IRC5Controller=? -1, SignalSource=SimulationProject 3637
EventTableTriggerIO 9180: Operator=0, IOValue=[0], IRC5Controller=? -1, SignalSource=SimulationProject 3637
EventTableTriggerIO 9181: Operator=0, IOValue=[0], IRC5Controller=? -1, SignalSource=SimulationProject 3637
EventTableTriggerIO 9182: Operator=0, IOValue=[0], IRC5Controller=? -1, SignalSource=SimulationProject 3637
EventTableTriggerIO 9183: Operator=0, IOValue=[0], IRC5Controller=? -1, SignalSource=SimulationProject 3637
EventTableTriggerIO 9184: Operator=0, IOValue=[0], IRC5Controller=? -1, SignalSource=SimulationProject 3637
EventTableTriggerIO 9185: Operator=0, IOValue=[0], IRC5Controller=? -1, SignalSource=SimulationProject 3637
EventTableTriggerIO 9186: Operator=0, IOValue=[0], IRC5Controller=? -1, SignalSource=SimulationProject 3637
EventTableTriggerIO 9187: Operator=0, IOValue=[1], IRC5Controller=? -1, SignalSource=SimulationProject 3637
EventTableTriggerIO 9188: Operator=0, IOValue=[1], IRC5Controller=? -1, SignalSource=SimulationProject 3637
EventTableTriggerIO 9189: Operator=0, IOValue=[1], IRC5Controller=? -1, SignalSource=SimulationProject 3637
EventTableTriggerIO 9190: Operator=0, IOValue=[1], IRC5Controller=? -1, SignalSource=SimulationProject 3637
EventTableTriggerIO 9191: Operator=0, IOValue=[1], IRC5Controller=? -1, SignalSource=SimulationProject 3637
EventTableTriggerIO 9192: Operator=0, IOValue=[1], IRC5Controller=? -1, SignalSource=SimulationProject 3637
EventTableTriggerIO 9193: Operator=0, IOValue=[1], IRC5Controller=? -1, SignalSource=SimulationProject 3637
EventTableTriggerIO 9194: Operator=0, IOValue=[0], IRC5Controller=? -1, SignalSource=SimulationProject 3637
EventTableTriggerIO 9195: Operator=0, IOValue=[0], IRC5Controller=? -1, SignalSource=SimulationProject 3637
EventTableTriggerIO 9196: Operator=0, IOValue=[0], IRC5Controller=? -1, SignalSource=SimulationProject 3637
EventTableTriggerIO 9197: Operator=0, IOValue=[0], IRC5Controller=? -1, SignalSource=SimulationProject 3637
EventTableTriggerIO 9198: Operator=0, IOValue=[0], IRC5Controller=? -1, SignalSource=SimulationProject 3637
EventTableTriggerIO 9199: Operator=0, IOValue=[0], IRC5Controller=? -1, SignalSource=SimulationProject 3637
EventTableTriggerIO 9200: Operator=0, IOValue=[0], IRC5Controller=? -1, SignalSource=SimulationProject 3637
EventTableTriggerIO 9201: Operator=0, IOValue=[1], IRC5Controller=? -1, SignalSource=SimulationProject 3637
EventTableTriggerIO 9202: Operator=0, IOValue=[1], IRC5Controller=? -1, SignalSource=SimulationProject 3637
EventTableTriggerIO 9203: Operator=0, IOValue=[1], IRC5Controller=? -1, SignalSource=SimulationProject 3637
EventTableTriggerIO 9204: Operator=0, IOValue=[1], IRC5Controller=? -1, SignalSource=SimulationProject 3637
EventTableTriggerIO 9205: Operator=0, IOValue=[1], IRC5Controller=? -1, SignalSource=SimulationProject 3637
EventTableTriggerIO 9206: Operator=0, IOValue=[1], IRC5Controller=? -1, SignalSource=SimulationProject 3637
EventTableTriggerIO 9207: Operator=0, IOValue=[1], IRC5Controller=? -1, SignalSource=SimulationProject 3637
EventTableTriggerIO 9208: Operator=0, IOValue=[0], IRC5Controller=? -1, SignalSource=SimulationProject 3637
EventTableTriggerIO 9209: Operator=0, IOValue=[0], IRC5Controller=? -1, SignalSource=SimulationProject 3637
EventTableTriggerIO 9210: Operator=0, IOValue=[0], IRC5Controller=? -1, SignalSource=SimulationProject 3637
EventTableTriggerIO 9211: Operator=0, IOValue=[0], IRC5Controller=? -1, SignalSource=SimulationProject 3637
EventTableTriggerIO 9212: Operator=0, IOValue=[0], IRC5Controller=? -1, SignalSource=SimulationProject 3637
EventTableTriggerIO 9213: Operator=0, IOValue=[0], IRC5Controller=? -1, SignalSource=SimulationProject 3637
EventTableTriggerIO 9214: Operator=0, IOValue=[0], IRC5Controller=? -1, SignalSource=SimulationProject 3637
EventTableTriggerIO 9252: Operator=0, IOValue=[1], IRC5Controller=? -1, SignalSource=SimulationProject 3637
EventTableTriggerIO 9253: Operator=0, IOValue=[1], IRC5Controller=? -1, SignalSource=SimulationProject 3637
EventTableTriggerIO 9254: Operator=0, IOValue=[1], IRC5Controller=? -1, SignalSource=SimulationProject 3637
EventTableTriggerIO 9255: Operator=0, IOValue=[0], IRC5Controller=? -1, SignalSource=SimulationProject 3637
EventTableTriggerIO 9256: Operator=0, IOValue=[0], IRC5Controller=? -1, SignalSource=SimulationProject 3637
EventTableTriggerIO 9257: Operator=0, IOValue=[0], IRC5Controller=? -1, SignalSource=SimulationProject 3637
EventTableTriggerIO 9258: Operator=0, IOValue=[1], IRC5Controller=? -1, SignalSource=SimulationProject 3637
EventTableTriggerIO 9259: Operator=0, IOValue=[1], IRC5Controller=? -1, SignalSource=SimulationProject 3637
EventTableTriggerIO 9260: Operator=0, IOValue=[1], IRC5Controller=? -1, SignalSource=SimulationProject 3637
EventTableTriggerIO 9261: Operator=0, IOValue=[0], IRC5Controller=? -1, SignalSource=SimulationProject 3637
EventTableTriggerIO 9262: Operator=0, IOValue=[0], IRC5Controller=? -1, SignalSource=SimulationProject 3637
EventTableTriggerIO 9263: Operator=0, IOValue=[0], IRC5Controller=? -1, SignalSource=SimulationProject 3637
EventTableTriggerIO 9264: Operator=0, IOValue=[1], IRC5Controller=? -1, SignalSource=SimulationProject 3637
EventTableTriggerIO 9265: Operator=0, IOValue=[1], IRC5Controller=? -1, SignalSource=SimulationProject 3637
EventTableTriggerIO 9266: Operator=0, IOValue=[1], IRC5Controller=? -1, SignalSource=SimulationProject 3637
EventTableTriggerIO 9267: Operator=0, IOValue=[0], IRC5Controller=? -1, SignalSource=SimulationProject 3637
EventTableTriggerIO 9268: Operator=0, IOValue=[0], IRC5Controller=? -1, SignalSource=SimulationProject 3637
EventTableTriggerIO 9269: Operator=0, IOValue=[0], IRC5Controller=? -1, SignalSource=SimulationProject 3637
EventTableTriggerIO 9270: Operator=0, IOValue=[1], IRC5Controller=? -1, SignalSource=SimulationProject 3637
EventTableTriggerIO 9271: Operator=0, IOValue=[1], IRC5Controller=? -1, SignalSource=SimulationProject 3637
EventTableTriggerIO 9272: Operator=0, IOValue=[1], IRC5Controller=? -1, SignalSource=SimulationProject 3637
EventTableTriggerIO 9273: Operator=0, IOValue=[0], IRC5Controller=? -1, SignalSource=SimulationProject 3637
EventTableTriggerIO 9274: Operator=0, IOValue=[0], IRC5Controller=? -1, SignalSource=SimulationProject 3637
EventTableTriggerIO 9275: Operator=0, IOValue=[0], IRC5Controller=? -1, SignalSource=SimulationProject 3637
EventTableTriggerIO 9276: Operator=0, IOValue=[1], IRC5Controller=? -1, SignalSource=SimulationProject 3637
EventTableTriggerIO 9277: Operator=0, IOValue=[1], IRC5Controller=? -1, SignalSource=SimulationProject 3637
EventTableTriggerIO 9278: Operator=0, IOValue=[1], IRC5Controller=? -1, SignalSource=SimulationProject 3637
EventTableTriggerIO 9279: Operator=0, IOValue=[0], IRC5Controller=? -1, SignalSource=SimulationProject 3637
EventTableTriggerIO 9280: Operator=0, IOValue=[0], IRC5Controller=? -1, SignalSource=SimulationProject 3637
EventTableTriggerIO 9281: Operator=0, IOValue=[0], IRC5Controller=? -1, SignalSource=SimulationProject 3637
EventTableTriggerIO 9282: Operator=0, IOValue=[1], IRC5Controller=? -1, SignalSource=SimulationProject 3637
EventTableTriggerIO 9283: Operator=0, IOValue=[1], IRC5Controller=? -1, SignalSource=SimulationProject 3637
EventTableTriggerIO 9284: Operator=0, IOValue=[1], IRC5Controller=? -1, SignalSource=SimulationProject 3637
EventTableTriggerIO 9285: Operator=0, IOValue=[0], IRC5Controller=? -1, SignalSource=SimulationProject 3637
EventTableTriggerIO 9286: Operator=0, IOValue=[0], IRC5Controller=? -1, SignalSource=SimulationProject 3637
EventTableTriggerIO 9287: Operator=0, IOValue=[0], IRC5Controller=? -1, SignalSource=SimulationProject 3637
EventTableTriggerIO 9288: Operator=0, IOValue=[1], IRC5Controller=? -1, SignalSource=SimulationProject 3637
EventTableTriggerIO 9289: Operator=0, IOValue=[1], IRC5Controller=? -1, SignalSource=SimulationProject 3637
EventTableTriggerIO 9290: Operator=0, IOValue=[1], IRC5Controller=? -1, SignalSource=SimulationProject 3637
EventTableTriggerIO 9291: Operator=0, IOValue=[0], IRC5Controller=? -1, SignalSource=SimulationProject 3637
EventTableTriggerIO 9292: Operator=0, IOValue=[0], IRC5Controller=? -1, SignalSource=SimulationProject 3637
EventTableTriggerIO 9293: Operator=0, IOValue=[0], IRC5Controller=? -1, SignalSource=SimulationProject 3637
EventTableTriggerIO 9294: Operator=0, IOValue=[1], IRC5Controller=? -1, SignalSource=SimulationProject 3637
EventTableTriggerIO 9295: Operator=0, IOValue=[1], IRC5Controller=? -1, SignalSource=SimulationProject 3637
EventTableTriggerIO 9296: Operator=0, IOValue=[1], IRC5Controller=? -1, SignalSource=SimulationProject 3637
EventTableTriggerIO 9297: Operator=0, IOValue=[0], IRC5Controller=? -1, SignalSource=SimulationProject 3637
EventTableTriggerIO 9298: Operator=0, IOValue=[0], IRC5Controller=? -1, SignalSource=SimulationProject 3637
EventTableTriggerIO 9299: Operator=0, IOValue=[0], IRC5Controller=? -1, SignalSource=SimulationProject 3637
EventTableTriggerIO 9300: Operator=0, IOValue=[1], IRC5Controller=? -1, SignalSource=SimulationProject 3637
EventTableTriggerIO 9301: Operator=0, IOValue=[1], IRC5Controller=? -1, SignalSource=SimulationProject 3637
EventTableTriggerIO 9302: Operator=0, IOValue=[1], IRC5Controller=? -1, SignalSource=SimulationProject 3637
EventTableTriggerIO 9303: Operator=0, IOValue=[0], IRC5Controller=? -1, SignalSource=SimulationProject 3637
EventTableTriggerIO 9304: Operator=0, IOValue=[0], IRC5Controller=? -1, SignalSource=SimulationProject 3637
EventTableTriggerIO 9305: Operator=0, IOValue=[0], IRC5Controller=? -1, SignalSource=SimulationProject 3637
EventTableTriggerIO 9306: Operator=0, IOValue=[1], IRC5Controller=? -1, SignalSource=SimulationProject 3637
EventTableTriggerIO 9307: Operator=0, IOValue=[1], IRC5Controller=? -1, SignalSource=SimulationProject 3637
EventTableTriggerIO 9308: Operator=0, IOValue=[1], IRC5Controller=? -1, SignalSource=SimulationProject 3637
EventTableTriggerIO 9309: Operator=0, IOValue=[0], IRC5Controller=? -1, SignalSource=SimulationProject 3637
EventTableTriggerIO 9310: Operator=0, IOValue=[0], IRC5Controller=? -1, SignalSource=SimulationProject 3637
EventTableTriggerIO 9311: Operator=0, IOValue=[0], IRC5Controller=? -1, SignalSource=SimulationProject 3637
EventTableTriggerIO 9331: Operator=0, IOValue=[1], IRC5Controller=? -1, SignalSource=SimulationProject 3637
EventTableTriggerIO 9332: Operator=0, IOValue=[0], IRC5Controller=? -1, SignalSource=SimulationProject 3637
EventTableTriggerIO 9333: Operator=0, IOValue=[1], IRC5Controller=? -1, SignalSource=SimulationProject 3637
EventTableTriggerIO 9334: Operator=0, IOValue=[0], IRC5Controller=? -1, SignalSource=SimulationProject 3637
EventTableTriggerIO 9335: Operator=0, IOValue=[1], IRC5Controller=? -1, SignalSource=SimulationProject 3637
EventTableTriggerIO 9336: Operator=0, IOValue=[0], IRC5Controller=? -1, SignalSource=SimulationProject 3637
EventTableTriggerIO 9337: Operator=0, IOValue=[1], IRC5Controller=? -1, SignalSource=SimulationProject 3637
EventTableTriggerIO 9338: Operator=0, IOValue=[0], IRC5Controller=? -1, SignalSource=SimulationProject 3637
EventTableTriggerIO 9339: Operator=0, IOValue=[1], IRC5Controller=? -1, SignalSource=SimulationProject 3637
EventTableTriggerIO 9340: Operator=0, IOValue=[0], IRC5Controller=? -1, SignalSource=SimulationProject 3637
EventTableTriggerIO 9341: Operator=0, IOValue=[1], IRC5Controller=? -1, SignalSource=SimulationProject 3637
EventTableTriggerIO 9342: Operator=0, IOValue=[0], IRC5Controller=? -1, SignalSource=SimulationProject 3637
EventTableTriggerIO 9343: Operator=0, IOValue=[1], IRC5Controller=? -1, SignalSource=SimulationProject 3637
EventTableTriggerIO 9344: Operator=0, IOValue=[0], IRC5Controller=? -1, SignalSource=SimulationProject 3637
EventTableTriggerIO 9345: Operator=0, IOValue=[1], IRC5Controller=? -1, SignalSource=SimulationProject 3637
EventTableTriggerIO 9346: Operator=0, IOValue=[0], IRC5Controller=? -1, SignalSource=SimulationProject 3637
EventTableTriggerIO 9347: Operator=0, IOValue=[1], IRC5Controller=? -1, SignalSource=SimulationProject 3637
EventTableTriggerIO 9348: Operator=0, IOValue=[0], IRC5Controller=? -1, SignalSource=SimulationProject 3637
EventTableTriggerIO 9349: Operator=0, IOValue=[1], IRC5Controller=? -1, SignalSource=SimulationProject 3637
EventTableTriggerIO 9350: Operator=0, IOValue=[0], IRC5Controller=? -1, SignalSource=SimulationProject 3637
EventTableTriggerIO 9953: Operator=0, IOValue=[1], IRC5Controller=? -1, SignalSource=SimulationProject 3637
EventTableTriggerIO 9954: Operator=0, IOValue=[1], IRC5Controller=? -1, SignalSource=SimulationProject 3637
EventTableTriggerIO 9955: Operator=0, IOValue=[0], IRC5Controller=? -1, SignalSource=SimulationProject 3637
EventTableTriggerIO 9956: Operator=0, IOValue=[0], IRC5Controller=? -1, SignalSource=SimulationProject 3637
EventTableTriggerIO 9957: Operator=0, IOValue=[1], IRC5Controller=? -1, SignalSource=SimulationProject 3637
EventTableTriggerIO 9958: Operator=0, IOValue=[1], IRC5Controller=? -1, SignalSource=SimulationProject 3637
EventTableTriggerIO 9959: Operator=0, IOValue=[0], IRC5Controller=? -1, SignalSource=SimulationProject 3637
EventTableTriggerIO 9960: Operator=0, IOValue=[0], IRC5Controller=? -1, SignalSource=SimulationProject 3637
EventTableTriggerIO 9961: Operator=0, IOValue=[1], IRC5Controller=? -1, SignalSource=SimulationProject 3637
EventTableTriggerIO 9962: Operator=0, IOValue=[1], IRC5Controller=? -1, SignalSource=SimulationProject 3637
EventTableTriggerIO 9963: Operator=0, IOValue=[0], IRC5Controller=? -1, SignalSource=SimulationProject 3637
EventTableTriggerIO 9964: Operator=0, IOValue=[0], IRC5Controller=? -1, SignalSource=SimulationProject 3637
EventTableTriggerIO 9965: Operator=0, IOValue=[1], IRC5Controller=? -1, SignalSource=SimulationProject 3637
EventTableTriggerIO 9966: Operator=0, IOValue=[1], IRC5Controller=? -1, SignalSource=SimulationProject 3637
EventTableTriggerIO 9967: Operator=0, IOValue=[0], IRC5Controller=? -1, SignalSource=SimulationProject 3637
EventTableTriggerIO 9968: Operator=0, IOValue=[0], IRC5Controller=? -1, SignalSource=SimulationProject 3637
EventTableTriggerIO 9969: Operator=0, IOValue=[1], IRC5Controller=? -1, SignalSource=SimulationProject 3637
EventTableTriggerIO 9970: Operator=0, IOValue=[1], IRC5Controller=? -1, SignalSource=SimulationProject 3637
EventTableTriggerIO 9971: Operator=0, IOValue=[0], IRC5Controller=? -1, SignalSource=SimulationProject 3637
EventTableTriggerIO 9972: Operator=0, IOValue=[0], IRC5Controller=? -1, SignalSource=SimulationProject 3637
EventTableTriggerIO 9973: Operator=0, IOValue=[1], IRC5Controller=? -1, SignalSource=SimulationProject 3637
EventTableTriggerIO 9974: Operator=0, IOValue=[1], IRC5Controller=? -1, SignalSource=SimulationProject 3637
EventTableTriggerIO 9975: Operator=0, IOValue=[0], IRC5Controller=? -1, SignalSource=SimulationProject 3637
EventTableTriggerIO 9976: Operator=0, IOValue=[0], IRC5Controller=? -1, SignalSource=SimulationProject 3637
EventTableTriggerIO 9977: Operator=0, IOValue=[1], IRC5Controller=? -1, SignalSource=SimulationProject 3637
EventTableTriggerIO 9978: Operator=0, IOValue=[1], IRC5Controller=? -1, SignalSource=SimulationProject 3637
EventTableTriggerIO 9979: Operator=0, IOValue=[0], IRC5Controller=? -1, SignalSource=SimulationProject 3637
EventTableTriggerIO 9980: Operator=0, IOValue=[0], IRC5Controller=? -1, SignalSource=SimulationProject 3637
EventTableTriggerIO 9981: Operator=0, IOValue=[1], IRC5Controller=? -1, SignalSource=SimulationProject 3637
EventTableTriggerIO 9982: Operator=0, IOValue=[1], IRC5Controller=? -1, SignalSource=SimulationProject 3637
EventTableTriggerIO 9983: Operator=0, IOValue=[0], IRC5Controller=? -1, SignalSource=SimulationProject 3637
EventTableTriggerIO 9984: Operator=0, IOValue=[0], IRC5Controller=? -1, SignalSource=SimulationProject 3637
EventTableTriggerIO 9985: Operator=0, IOValue=[1], IRC5Controller=? -1, SignalSource=SimulationProject 3637
EventTableTriggerIO 9986: Operator=0, IOValue=[1], IRC5Controller=? -1, SignalSource=SimulationProject 3637
EventTableTriggerIO 9987: Operator=0, IOValue=[0], IRC5Controller=? -1, SignalSource=SimulationProject 3637
EventTableTriggerIO 9988: Operator=0, IOValue=[0], IRC5Controller=? -1, SignalSource=SimulationProject 3637
EventTableTriggerIO 9989: Operator=0, IOValue=[1], IRC5Controller=? -1, SignalSource=SimulationProject 3637
EventTableTriggerIO 9990: Operator=0, IOValue=[1], IRC5Controller=? -1, SignalSource=SimulationProject 3637
EventTableTriggerIO 9991: Operator=0, IOValue=[0], IRC5Controller=? -1, SignalSource=SimulationProject 3637
EventTableTriggerIO 9992: Operator=0, IOValue=[0], IRC5Controller=? -1, SignalSource=SimulationProject 3637
EventTableEntry 9996: ActivationMode=2, Cyclic=false, Group=, Trigger=doWheelTool_L 9997, Actions=[EventTableActionAttach 9998], Comment=
EventTableTriggerIO 9997: Operator=0, IOValue=[1], IRC5Controller=? -1, SignalSource=SimulationProject 3637
EventTableActionAttach 9998: MountObject=false, FlangeIndext=0, FindNearest=false, AttachmentParent=IRB6660_100_335__01_L 3595, AttachmentChild=WheelTool_L 5987, Offset=[X=1, Y=0, Z=0, W=0, X=0, Y=1, Z=0, W=0, X=0, Y=0, Z=1, W=0, X=0, Y=0, Z=0, W=1]
EventTableEntry 9999: ActivationMode=2, Cyclic=false, Group=, Trigger=doWheelTool_L 10000, Actions=[EventTableActionDetach 10001], Comment=
EventTableTriggerIO 10000: Operator=0, IOValue=[0], IRC5Controller=? -1, SignalSource=SimulationProject 3637
EventTableActionDetach 10001: AttachmentParent=IRB6660_100_335__01_L 3595, AttachmentChild=WheelTool_L 5987
EventTableEntry 10002: ActivationMode=2, Cyclic=false, Group=, Trigger=doWheel_L 10003, Actions=[EventTableActionAttach 10004], Comment=
EventTableTriggerIO 10003: Operator=0, IOValue=[1], IRC5Controller=? -1, SignalSource=SimulationProject 3637
EventTableActionAttach 10004: MountObject=false, FlangeIndext=0, FindNearest=true, AttachmentParent=WheelTool_L 5987, AttachmentChild=? -1, Offset=[X=1, Y=0, Z=0, W=0, X=0, Y=1, Z=0, W=0, X=0, Y=0, Z=1, W=0, X=0, Y=0, Z=0, W=1]
EventTableEntry 10005: ActivationMode=2, Cyclic=false, Group=, Trigger=doWheel_L 10006, Actions=[EventTableActionDetach 10007], Comment=
EventTableTriggerIO 10006: Operator=0, IOValue=[0], IRC5Controller=? -1, SignalSource=SimulationProject 3637
EventTableActionDetach 10007: AttachmentParent=WheelTool_L 5987, AttachmentChild=? -1
EventTableTriggerIO 10008: Operator=0, IOValue=[1], IRC5Controller=? -1, SignalSource=SimulationProject 3637
EventTableTriggerIO 10009: Operator=0, IOValue=[1], IRC5Controller=? -1, SignalSource=SimulationProject 3637
EventTableTriggerIO 10010: Operator=0, IOValue=[1], IRC5Controller=? -1, SignalSource=SimulationProject 3637
EventTableTriggerIO 10011: Operator=0, IOValue=[0], IRC5Controller=? -1, SignalSource=SimulationProject 3637
EventTableTriggerIO 10012: Operator=0, IOValue=[0], IRC5Controller=? -1, SignalSource=SimulationProject 3637
EventTableTriggerIO 10013: Operator=0, IOValue=[0], IRC5Controller=? -1, SignalSource=SimulationProject 3637
EventTableTriggerIO 10014: Operator=0, IOValue=[1], IRC5Controller=? -1, SignalSource=SimulationProject 3637
EventTableTriggerIO 10015: Operator=0, IOValue=[1], IRC5Controller=? -1, SignalSource=SimulationProject 3637
EventTableTriggerIO 10016: Operator=0, IOValue=[1], IRC5Controller=? -1, SignalSource=SimulationProject 3637
EventTableTriggerIO 10017: Operator=0, IOValue=[0], IRC5Controller=? -1, SignalSource=SimulationProject 3637
EventTableTriggerIO 10018: Operator=0, IOValue=[0], IRC5Controller=? -1, SignalSource=SimulationProject 3637
EventTableTriggerIO 10019: Operator=0, IOValue=[0], IRC5Controller=? -1, SignalSource=SimulationProject 3637
EventTableTriggerIO 10020: Operator=0, IOValue=[1], IRC5Controller=? -1, SignalSource=SimulationProject 3637
EventTableTriggerIO 10021: Operator=0, IOValue=[1], IRC5Controller=? -1, SignalSource=SimulationProject 3637
EventTableTriggerIO 10022: Operator=0, IOValue=[1], IRC5Controller=? -1, SignalSource=SimulationProject 3637
EventTableTriggerIO 10023: Operator=0, IOValue=[0], IRC5Controller=? -1, SignalSource=SimulationProject 3637
EventTableTriggerIO 10024: Operator=0, IOValue=[0], IRC5Controller=? -1, SignalSource=SimulationProject 3637
EventTableTriggerIO 10025: Operator=0, IOValue=[0], IRC5Controller=? -1, SignalSource=SimulationProject 3637
EventTableTriggerIO 10026: Operator=0, IOValue=[1], IRC5Controller=? -1, SignalSource=SimulationProject 3637
EventTableTriggerIO 10027: Operator=0, IOValue=[1], IRC5Controller=? -1, SignalSource=SimulationProject 3637
EventTableTriggerIO 10028: Operator=0, IOValue=[1], IRC5Controller=? -1, SignalSource=SimulationProject 3637
EventTableTriggerIO 10029: Operator=0, IOValue=[0], IRC5Controller=? -1, SignalSource=SimulationProject 3637
EventTableTriggerIO 10030: Operator=0, IOValue=[0], IRC5Controller=? -1, SignalSource=SimulationProject 3637
EventTableTriggerIO 10031: Operator=0, IOValue=[0], IRC5Controller=? -1, SignalSource=SimulationProject 3637
EventTableTriggerIO 10032: Operator=0, IOValue=[1], IRC5Controller=? -1, SignalSource=SimulationProject 3637
EventTableTriggerIO 10033: Operator=0, IOValue=[1], IRC5Controller=? -1, SignalSource=SimulationProject 3637
EventTableTriggerIO 10034: Operator=0, IOValue=[1], IRC5Controller=? -1, SignalSource=SimulationProject 3637
EventTableTriggerIO 10035: Operator=0, IOValue=[0], IRC5Controller=? -1, SignalSource=SimulationProject 3637
EventTableTriggerIO 10036: Operator=0, IOValue=[0], IRC5Controller=? -1, SignalSource=SimulationProject 3637
EventTableTriggerIO 10037: Operator=0, IOValue=[0], IRC5Controller=? -1, SignalSource=SimulationProject 3637
EventTableTriggerIO 10038: Operator=0, IOValue=[1], IRC5Controller=? -1, SignalSource=SimulationProject 3637
EventTableTriggerIO 10039: Operator=0, IOValue=[1], IRC5Controller=? -1, SignalSource=SimulationProject 3637
EventTableTriggerIO 10040: Operator=0, IOValue=[1], IRC5Controller=? -1, SignalSource=SimulationProject 3637
EventTableTriggerIO 10041: Operator=0, IOValue=[0], IRC5Controller=? -1, SignalSource=SimulationProject 3637
EventTableTriggerIO 10042: Operator=0, IOValue=[0], IRC5Controller=? -1, SignalSource=SimulationProject 3637
EventTableTriggerIO 10043: Operator=0, IOValue=[0], IRC5Controller=? -1, SignalSource=SimulationProject 3637
EventTableTriggerIO 10044: Operator=0, IOValue=[1], IRC5Controller=? -1, SignalSource=SimulationProject 3637
EventTableTriggerIO 10045: Operator=0, IOValue=[1], IRC5Controller=? -1, SignalSource=SimulationProject 3637
EventTableTriggerIO 10046: Operator=0, IOValue=[1], IRC5Controller=? -1, SignalSource=SimulationProject 3637
EventTableTriggerIO 10047: Operator=0, IOValue=[0], IRC5Controller=? -1, SignalSource=SimulationProject 3637
EventTableTriggerIO 10048: Operator=0, IOValue=[0], IRC5Controller=? -1, SignalSource=SimulationProject 3637
EventTableTriggerIO 10049: Operator=0, IOValue=[0], IRC5Controller=? -1, SignalSource=SimulationProject 3637
EventTableTriggerIO 10050: Operator=0, IOValue=[1], IRC5Controller=? -1, SignalSource=SimulationProject 3637
EventTableTriggerIO 10051: Operator=0, IOValue=[1], IRC5Controller=? -1, SignalSource=SimulationProject 3637
EventTableTriggerIO 10052: Operator=0, IOValue=[1], IRC5Controller=? -1, SignalSource=SimulationProject 3637
EventTableTriggerIO 10053: Operator=0, IOValue=[0], IRC5Controller=? -1, SignalSource=SimulationProject 3637
EventTableTriggerIO 10054: Operator=0, IOValue=[0], IRC5Controller=? -1, SignalSource=SimulationProject 3637
EventTableTriggerIO 10055: Operator=0, IOValue=[0], IRC5Controller=? -1, SignalSource=SimulationProject 3637
EventTableTriggerIO 10056: Operator=0, IOValue=[1], IRC5Controller=? -1, SignalSource=SimulationProject 3637
EventTableTriggerIO 10057: Operator=0, IOValue=[1], IRC5Controller=? -1, SignalSource=SimulationProject 3637
